REGION Network 10: DIa5
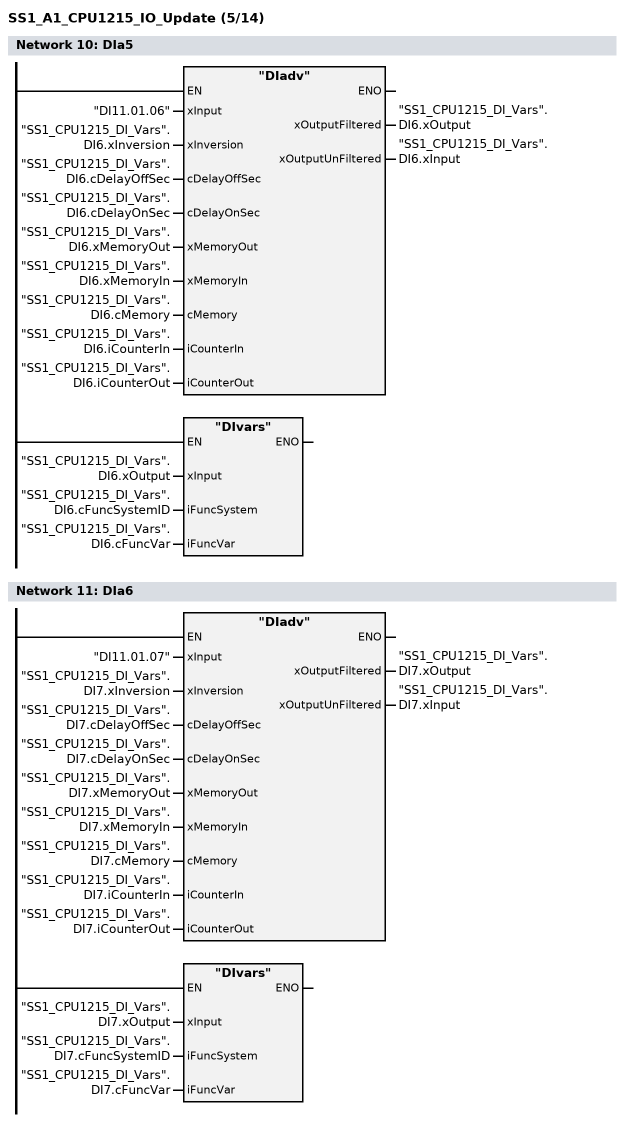
   RUNG wire#powerrail
      "DIadv"(xInput := "DI11.01.06", xInversion := "SS1_CPU1215_DI_Vars".DI6.xInversion, cDelayOffSec := "SS1_CPU1215_DI_Vars".DI6.cDelayOffSec, cDelayOnSec := "SS1_CPU1215_DI_Vars".DI6.cDelayOnSec, xMemoryOut := "SS1_CPU1215_DI_Vars".DI6.xMemoryOut, xMemoryIn := "SS1_CPU1215_DI_Vars".DI6.xMemoryIn, cMemory := "SS1_CPU1215_DI_Vars".DI6.cMemory, xOutputFiltered => "SS1_CPU1215_DI_Vars".DI6.xOutput, xOutputUnFiltered => "SS1_CPU1215_DI_Vars".DI6.xInput, iCounterIn := "SS1_CPU1215_DI_Vars".DI6.iCounterIn, iCounterOut := "SS1_CPU1215_DI_Vars".DI6.iCounterOut)
   END_RUNG
   RUNG wire#powerrail
      "DIvars"(xInput := "SS1_CPU1215_DI_Vars".DI6.xOutput, iFuncSystem := "SS1_CPU1215_DI_Vars".DI6.cFuncSystemID, iFuncVar := "SS1_CPU1215_DI_Vars".DI6.cFuncVar)
   END_RUNG
   // the same network as SCL:
   "DIadv"(xInput := "DI11.01.06",
           xInversion := "SS1_CPU1215_DI_Vars".DI6.xInversion,
           cDelayOffSec := "SS1_CPU1215_DI_Vars".DI6.cDelayOffSec,
           cDelayOnSec := "SS1_CPU1215_DI_Vars".DI6.cDelayOnSec,
           xMemoryOut := "SS1_CPU1215_DI_Vars".DI6.xMemoryOut,
           xMemoryIn := "SS1_CPU1215_DI_Vars".DI6.xMemoryIn,
           cMemory := "SS1_CPU1215_DI_Vars".DI6.cMemory,
           iCounterIn := "SS1_CPU1215_DI_Vars".DI6.iCounterIn,
           iCounterOut := "SS1_CPU1215_DI_Vars".DI6.iCounterOut,
           xOutputFiltered => "SS1_CPU1215_DI_Vars".DI6.xOutput,
           xOutputUnFiltered => "SS1_CPU1215_DI_Vars".DI6.xInput);
   "DIvars"(xInput := "SS1_CPU1215_DI_Vars".DI6.xOutput,
            iFuncSystem := "SS1_CPU1215_DI_Vars".DI6.cFuncSystemID,
            iFuncVar := "SS1_CPU1215_DI_Vars".DI6.cFuncVar);
END_REGION

REGION Network 11: DIa6
   RUNG wire#powerrail
      "DIadv"(xInput := "DI11.01.07", xInversion := "SS1_CPU1215_DI_Vars".DI7.xInversion, cDelayOffSec := "SS1_CPU1215_DI_Vars".DI7.cDelayOffSec, cDelayOnSec := "SS1_CPU1215_DI_Vars".DI7.cDelayOnSec, xMemoryOut := "SS1_CPU1215_DI_Vars".DI7.xMemoryOut, xMemoryIn := "SS1_CPU1215_DI_Vars".DI7.xMemoryIn, cMemory := "SS1_CPU1215_DI_Vars".DI7.cMemory, xOutputFiltered => "SS1_CPU1215_DI_Vars".DI7.xOutput, xOutputUnFiltered => "SS1_CPU1215_DI_Vars".DI7.xInput, iCounterIn := "SS1_CPU1215_DI_Vars".DI7.iCounterIn, iCounterOut := "SS1_CPU1215_DI_Vars".DI7.iCounterOut)
   END_RUNG
   RUNG wire#powerrail
      "DIvars"(xInput := "SS1_CPU1215_DI_Vars".DI7.xOutput, iFuncSystem := "SS1_CPU1215_DI_Vars".DI7.cFuncSystemID, iFuncVar := "SS1_CPU1215_DI_Vars".DI7.cFuncVar)
   END_RUNG
   // the same network as SCL:
   "DIadv"(xInput := "DI11.01.07",
           xInversion := "SS1_CPU1215_DI_Vars".DI7.xInversion,
           cDelayOffSec := "SS1_CPU1215_DI_Vars".DI7.cDelayOffSec,
           cDelayOnSec := "SS1_CPU1215_DI_Vars".DI7.cDelayOnSec,
           xMemoryOut := "SS1_CPU1215_DI_Vars".DI7.xMemoryOut,
           xMemoryIn := "SS1_CPU1215_DI_Vars".DI7.xMemoryIn,
           cMemory := "SS1_CPU1215_DI_Vars".DI7.cMemory,
           iCounterIn := "SS1_CPU1215_DI_Vars".DI7.iCounterIn,
           iCounterOut := "SS1_CPU1215_DI_Vars".DI7.iCounterOut,
           xOutputFiltered => "SS1_CPU1215_DI_Vars".DI7.xOutput,
           xOutputUnFiltered => "SS1_CPU1215_DI_Vars".DI7.xInput);
   "DIvars"(xInput := "SS1_CPU1215_DI_Vars".DI7.xOutput,
            iFuncSystem := "SS1_CPU1215_DI_Vars".DI7.cFuncSystemID,
            iFuncVar := "SS1_CPU1215_DI_Vars".DI7.cFuncVar);
END_REGION

REGION Network 12: DIa7 / DI01.1.08 EDP під охороною
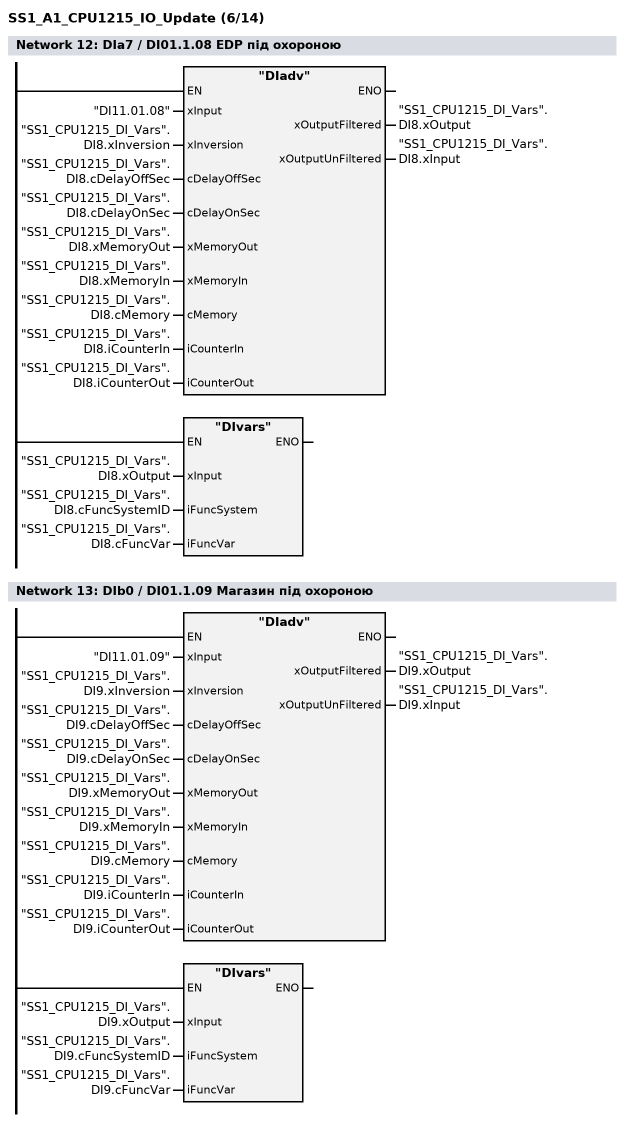
   RUNG wire#powerrail
      "DIadv"(xInput := "DI11.01.08", xInversion := "SS1_CPU1215_DI_Vars".DI8.xInversion, cDelayOffSec := "SS1_CPU1215_DI_Vars".DI8.cDelayOffSec, cDelayOnSec := "SS1_CPU1215_DI_Vars".DI8.cDelayOnSec, xMemoryOut := "SS1_CPU1215_DI_Vars".DI8.xMemoryOut, xMemoryIn := "SS1_CPU1215_DI_Vars".DI8.xMemoryIn, cMemory := "SS1_CPU1215_DI_Vars".DI8.cMemory, iCounterIn := "SS1_CPU1215_DI_Vars".DI8.iCounterIn, iCounterOut := "SS1_CPU1215_DI_Vars".DI8.iCounterOut, xOutputFiltered => "SS1_CPU1215_DI_Vars".DI8.xOutput, xOutputUnFiltered => "SS1_CPU1215_DI_Vars".DI8.xInput)
   END_RUNG
   RUNG wire#powerrail
      "DIvars"(xInput := "SS1_CPU1215_DI_Vars".DI8.xOutput, iFuncSystem := "SS1_CPU1215_DI_Vars".DI8.cFuncSystemID, iFuncVar := "SS1_CPU1215_DI_Vars".DI8.cFuncVar)
   END_RUNG
   // the same network as SCL:
   "DIadv"(xInput := "DI11.01.08",
           xInversion := "SS1_CPU1215_DI_Vars".DI8.xInversion,
           cDelayOffSec := "SS1_CPU1215_DI_Vars".DI8.cDelayOffSec,
           cDelayOnSec := "SS1_CPU1215_DI_Vars".DI8.cDelayOnSec,
           xMemoryOut := "SS1_CPU1215_DI_Vars".DI8.xMemoryOut,
           xMemoryIn := "SS1_CPU1215_DI_Vars".DI8.xMemoryIn,
           cMemory := "SS1_CPU1215_DI_Vars".DI8.cMemory,
           iCounterIn := "SS1_CPU1215_DI_Vars".DI8.iCounterIn,
           iCounterOut := "SS1_CPU1215_DI_Vars".DI8.iCounterOut,
           xOutputFiltered => "SS1_CPU1215_DI_Vars".DI8.xOutput,
           xOutputUnFiltered => "SS1_CPU1215_DI_Vars".DI8.xInput);
   "DIvars"(xInput := "SS1_CPU1215_DI_Vars".DI8.xOutput,
            iFuncSystem := "SS1_CPU1215_DI_Vars".DI8.cFuncSystemID,
            iFuncVar := "SS1_CPU1215_DI_Vars".DI8.cFuncVar);
END_REGION

REGION Network 13: DIb0 / DI01.1.09 Магазин під охороною
   RUNG wire#powerrail
      "DIadv"(xInput := "DI11.01.09", xInversion := "SS1_CPU1215_DI_Vars".DI9.xInversion, cDelayOffSec := "SS1_CPU1215_DI_Vars".DI9.cDelayOffSec, cDelayOnSec := "SS1_CPU1215_DI_Vars".DI9.cDelayOnSec, xMemoryOut := "SS1_CPU1215_DI_Vars".DI9.xMemoryOut, xMemoryIn := "SS1_CPU1215_DI_Vars".DI9.xMemoryIn, cMemory := "SS1_CPU1215_DI_Vars".DI9.cMemory, xOutputFiltered => "SS1_CPU1215_DI_Vars".DI9.xOutput, xOutputUnFiltered => "SS1_CPU1215_DI_Vars".DI9.xInput, iCounterIn := "SS1_CPU1215_DI_Vars".DI9.iCounterIn, iCounterOut := "SS1_CPU1215_DI_Vars".DI9.iCounterOut)
   END_RUNG
   RUNG wire#powerrail
      "DIvars"(xInput := "SS1_CPU1215_DI_Vars".DI9.xOutput, iFuncSystem := "SS1_CPU1215_DI_Vars".DI9.cFuncSystemID, iFuncVar := "SS1_CPU1215_DI_Vars".DI9.cFuncVar)
   END_RUNG
   // the same network as SCL:
   "DIadv"(xInput := "DI11.01.09",
           xInversion := "SS1_CPU1215_DI_Vars".DI9.xInversion,
           cDelayOffSec := "SS1_CPU1215_DI_Vars".DI9.cDelayOffSec,
           cDelayOnSec := "SS1_CPU1215_DI_Vars".DI9.cDelayOnSec,
           xMemoryOut := "SS1_CPU1215_DI_Vars".DI9.xMemoryOut,
           xMemoryIn := "SS1_CPU1215_DI_Vars".DI9.xMemoryIn,
           cMemory := "SS1_CPU1215_DI_Vars".DI9.cMemory,
           iCounterIn := "SS1_CPU1215_DI_Vars".DI9.iCounterIn,
           iCounterOut := "SS1_CPU1215_DI_Vars".DI9.iCounterOut,
           xOutputFiltered => "SS1_CPU1215_DI_Vars".DI9.xOutput,
           xOutputUnFiltered => "SS1_CPU1215_DI_Vars".DI9.xInput);
   "DIvars"(xInput := "SS1_CPU1215_DI_Vars".DI9.xOutput,
            iFuncSystem := "SS1_CPU1215_DI_Vars".DI9.cFuncSystemID,
            iFuncVar := "SS1_CPU1215_DI_Vars".DI9.cFuncVar);
END_REGION

REGION Network 14: DIb1 / DI01.1.10 Аварійний рівень загазованості
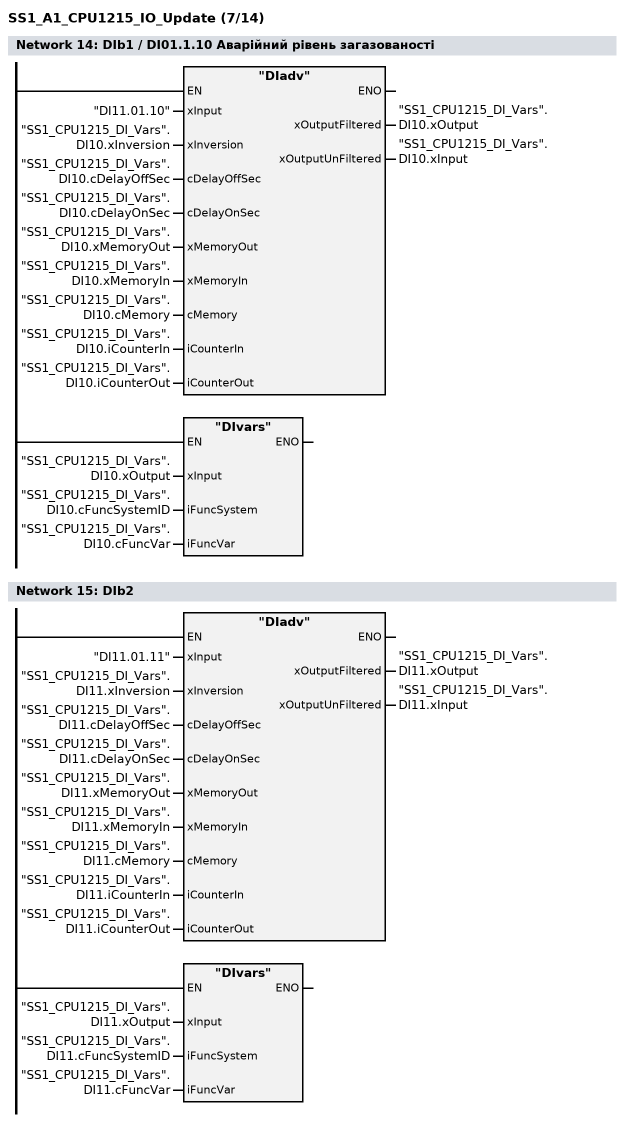
   RUNG wire#powerrail
      "DIadv"(xInput := "DI11.01.10", xInversion := "SS1_CPU1215_DI_Vars".DI10.xInversion, cDelayOffSec := "SS1_CPU1215_DI_Vars".DI10.cDelayOffSec, cDelayOnSec := "SS1_CPU1215_DI_Vars".DI10.cDelayOnSec, xMemoryOut := "SS1_CPU1215_DI_Vars".DI10.xMemoryOut, xMemoryIn := "SS1_CPU1215_DI_Vars".DI10.xMemoryIn, cMemory := "SS1_CPU1215_DI_Vars".DI10.cMemory, xOutputFiltered => "SS1_CPU1215_DI_Vars".DI10.xOutput, xOutputUnFiltered => "SS1_CPU1215_DI_Vars".DI10.xInput, iCounterIn := "SS1_CPU1215_DI_Vars".DI10.iCounterIn, iCounterOut := "SS1_CPU1215_DI_Vars".DI10.iCounterOut)
   END_RUNG
   RUNG wire#powerrail
      "DIvars"(xInput := "SS1_CPU1215_DI_Vars".DI10.xOutput, iFuncSystem := "SS1_CPU1215_DI_Vars".DI10.cFuncSystemID, iFuncVar := "SS1_CPU1215_DI_Vars".DI10.cFuncVar)
   END_RUNG
   // the same network as SCL:
   "DIadv"(xInput := "DI11.01.10",
           xInversion := "SS1_CPU1215_DI_Vars".DI10.xInversion,
           cDelayOffSec := "SS1_CPU1215_DI_Vars".DI10.cDelayOffSec,
           cDelayOnSec := "SS1_CPU1215_DI_Vars".DI10.cDelayOnSec,
           xMemoryOut := "SS1_CPU1215_DI_Vars".DI10.xMemoryOut,
           xMemoryIn := "SS1_CPU1215_DI_Vars".DI10.xMemoryIn,
           cMemory := "SS1_CPU1215_DI_Vars".DI10.cMemory,
           iCounterIn := "SS1_CPU1215_DI_Vars".DI10.iCounterIn,
           iCounterOut := "SS1_CPU1215_DI_Vars".DI10.iCounterOut,
           xOutputFiltered => "SS1_CPU1215_DI_Vars".DI10.xOutput,
           xOutputUnFiltered => "SS1_CPU1215_DI_Vars".DI10.xInput);
   "DIvars"(xInput := "SS1_CPU1215_DI_Vars".DI10.xOutput,
            iFuncSystem := "SS1_CPU1215_DI_Vars".DI10.cFuncSystemID,
            iFuncVar := "SS1_CPU1215_DI_Vars".DI10.cFuncVar);
END_REGION

REGION Network 15: DIb2
   RUNG wire#powerrail
      "DIadv"(xInput := "DI11.01.11", xInversion := "SS1_CPU1215_DI_Vars".DI11.xInversion, cDelayOffSec := "SS1_CPU1215_DI_Vars".DI11.cDelayOffSec, cDelayOnSec := "SS1_CPU1215_DI_Vars".DI11.cDelayOnSec, xMemoryOut := "SS1_CPU1215_DI_Vars".DI11.xMemoryOut, xMemoryIn := "SS1_CPU1215_DI_Vars".DI11.xMemoryIn, cMemory := "SS1_CPU1215_DI_Vars".DI11.cMemory, iCounterIn := "SS1_CPU1215_DI_Vars".DI11.iCounterIn, iCounterOut := "SS1_CPU1215_DI_Vars".DI11.iCounterOut, xOutputFiltered => "SS1_CPU1215_DI_Vars".DI11.xOutput, xOutputUnFiltered => "SS1_CPU1215_DI_Vars".DI11.xInput)
   END_RUNG
   RUNG wire#powerrail
      "DIvars"(xInput := "SS1_CPU1215_DI_Vars".DI11.xOutput, iFuncSystem := "SS1_CPU1215_DI_Vars".DI11.cFuncSystemID, iFuncVar := "SS1_CPU1215_DI_Vars".DI11.cFuncVar)
   END_RUNG
   // the same network as SCL:
   "DIadv"(xInput := "DI11.01.11",
           xInversion := "SS1_CPU1215_DI_Vars".DI11.xInversion,
           cDelayOffSec := "SS1_CPU1215_DI_Vars".DI11.cDelayOffSec,
           cDelayOnSec := "SS1_CPU1215_DI_Vars".DI11.cDelayOnSec,
           xMemoryOut := "SS1_CPU1215_DI_Vars".DI11.xMemoryOut,
           xMemoryIn := "SS1_CPU1215_DI_Vars".DI11.xMemoryIn,
           cMemory := "SS1_CPU1215_DI_Vars".DI11.cMemory,
           iCounterIn := "SS1_CPU1215_DI_Vars".DI11.iCounterIn,
           iCounterOut := "SS1_CPU1215_DI_Vars".DI11.iCounterOut,
           xOutputFiltered => "SS1_CPU1215_DI_Vars".DI11.xOutput,
           xOutputUnFiltered => "SS1_CPU1215_DI_Vars".DI11.xInput);
   "DIvars"(xInput := "SS1_CPU1215_DI_Vars".DI11.xOutput,
            iFuncSystem := "SS1_CPU1215_DI_Vars".DI11.cFuncSystemID,
            iFuncVar := "SS1_CPU1215_DI_Vars".DI11.cFuncVar);
END_REGION

REGION Network 16: DIb3
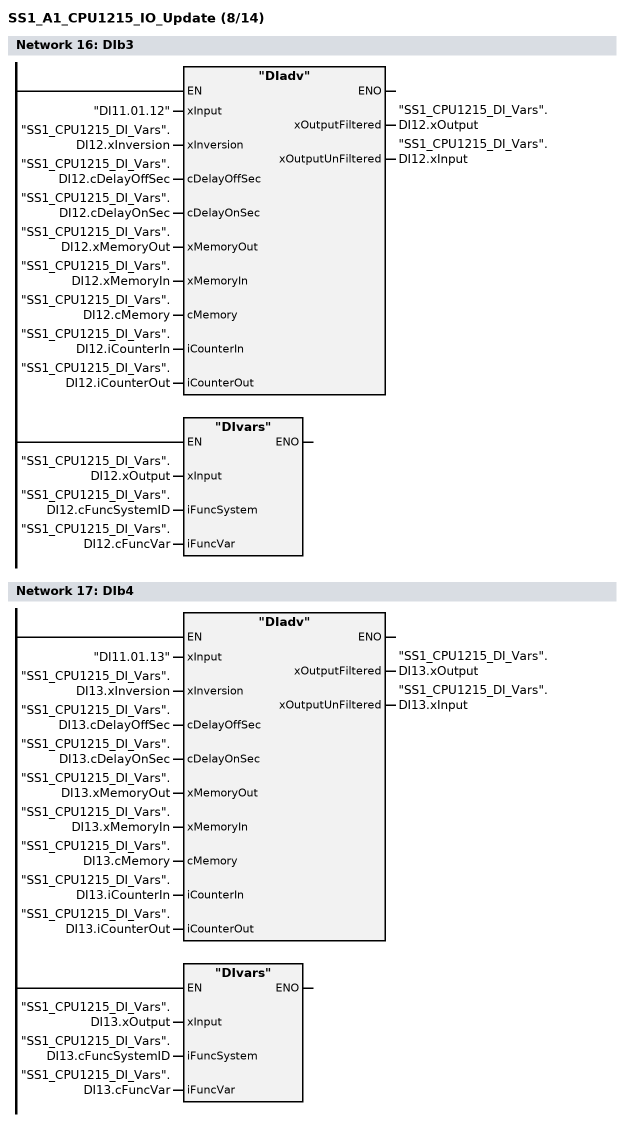
   RUNG wire#powerrail
      "DIadv"(xInput := "DI11.01.12", xInversion := "SS1_CPU1215_DI_Vars".DI12.xInversion, cDelayOffSec := "SS1_CPU1215_DI_Vars".DI12.cDelayOffSec, cDelayOnSec := "SS1_CPU1215_DI_Vars".DI12.cDelayOnSec, xMemoryOut := "SS1_CPU1215_DI_Vars".DI12.xMemoryOut, xMemoryIn := "SS1_CPU1215_DI_Vars".DI12.xMemoryIn, cMemory := "SS1_CPU1215_DI_Vars".DI12.cMemory, xOutputFiltered => "SS1_CPU1215_DI_Vars".DI12.xOutput, xOutputUnFiltered => "SS1_CPU1215_DI_Vars".DI12.xInput, iCounterIn := "SS1_CPU1215_DI_Vars".DI12.iCounterIn, iCounterOut := "SS1_CPU1215_DI_Vars".DI12.iCounterOut)
   END_RUNG
   RUNG wire#powerrail
      "DIvars"(xInput := "SS1_CPU1215_DI_Vars".DI12.xOutput, iFuncSystem := "SS1_CPU1215_DI_Vars".DI12.cFuncSystemID, iFuncVar := "SS1_CPU1215_DI_Vars".DI12.cFuncVar)
   END_RUNG
   // the same network as SCL:
   "DIadv"(xInput := "DI11.01.12",
           xInversion := "SS1_CPU1215_DI_Vars".DI12.xInversion,
           cDelayOffSec := "SS1_CPU1215_DI_Vars".DI12.cDelayOffSec,
           cDelayOnSec := "SS1_CPU1215_DI_Vars".DI12.cDelayOnSec,
           xMemoryOut := "SS1_CPU1215_DI_Vars".DI12.xMemoryOut,
           xMemoryIn := "SS1_CPU1215_DI_Vars".DI12.xMemoryIn,
           cMemory := "SS1_CPU1215_DI_Vars".DI12.cMemory,
           iCounterIn := "SS1_CPU1215_DI_Vars".DI12.iCounterIn,
           iCounterOut := "SS1_CPU1215_DI_Vars".DI12.iCounterOut,
           xOutputFiltered => "SS1_CPU1215_DI_Vars".DI12.xOutput,
           xOutputUnFiltered => "SS1_CPU1215_DI_Vars".DI12.xInput);
   "DIvars"(xInput := "SS1_CPU1215_DI_Vars".DI12.xOutput,
            iFuncSystem := "SS1_CPU1215_DI_Vars".DI12.cFuncSystemID,
            iFuncVar := "SS1_CPU1215_DI_Vars".DI12.cFuncVar);
END_REGION

REGION Network 17: DIb4
   RUNG wire#powerrail
      "DIadv"(xInput := "DI11.01.13", xInversion := "SS1_CPU1215_DI_Vars".DI13.xInversion, cDelayOffSec := "SS1_CPU1215_DI_Vars".DI13.cDelayOffSec, cDelayOnSec := "SS1_CPU1215_DI_Vars".DI13.cDelayOnSec, xMemoryOut := "SS1_CPU1215_DI_Vars".DI13.xMemoryOut, xMemoryIn := "SS1_CPU1215_DI_Vars".DI13.xMemoryIn, cMemory := "SS1_CPU1215_DI_Vars".DI13.cMemory, xOutputFiltered => "SS1_CPU1215_DI_Vars".DI13.xOutput, xOutputUnFiltered => "SS1_CPU1215_DI_Vars".DI13.xInput, iCounterIn := "SS1_CPU1215_DI_Vars".DI13.iCounterIn, iCounterOut := "SS1_CPU1215_DI_Vars".DI13.iCounterOut)
   END_RUNG
   RUNG wire#powerrail
      "DIvars"(xInput := "SS1_CPU1215_DI_Vars".DI13.xOutput, iFuncSystem := "SS1_CPU1215_DI_Vars".DI13.cFuncSystemID, iFuncVar := "SS1_CPU1215_DI_Vars".DI13.cFuncVar)
   END_RUNG
   // the same network as SCL:
   "DIadv"(xInput := "DI11.01.13",
           xInversion := "SS1_CPU1215_DI_Vars".DI13.xInversion,
           cDelayOffSec := "SS1_CPU1215_DI_Vars".DI13.cDelayOffSec,
           cDelayOnSec := "SS1_CPU1215_DI_Vars".DI13.cDelayOnSec,
           xMemoryOut := "SS1_CPU1215_DI_Vars".DI13.xMemoryOut,
           xMemoryIn := "SS1_CPU1215_DI_Vars".DI13.xMemoryIn,
           cMemory := "SS1_CPU1215_DI_Vars".DI13.cMemory,
           iCounterIn := "SS1_CPU1215_DI_Vars".DI13.iCounterIn,
           iCounterOut := "SS1_CPU1215_DI_Vars".DI13.iCounterOut,
           xOutputFiltered => "SS1_CPU1215_DI_Vars".DI13.xOutput,
           xOutputUnFiltered => "SS1_CPU1215_DI_Vars".DI13.xInput);
   "DIvars"(xInput := "SS1_CPU1215_DI_Vars".DI13.xOutput,
            iFuncSystem := "SS1_CPU1215_DI_Vars".DI13.cFuncSystemID,
            iFuncVar := "SS1_CPU1215_DI_Vars".DI13.cFuncVar);
END_REGION

REGION Network 18: DIb5 / DI01.1.14 Спрацювання охоронної сигналізації
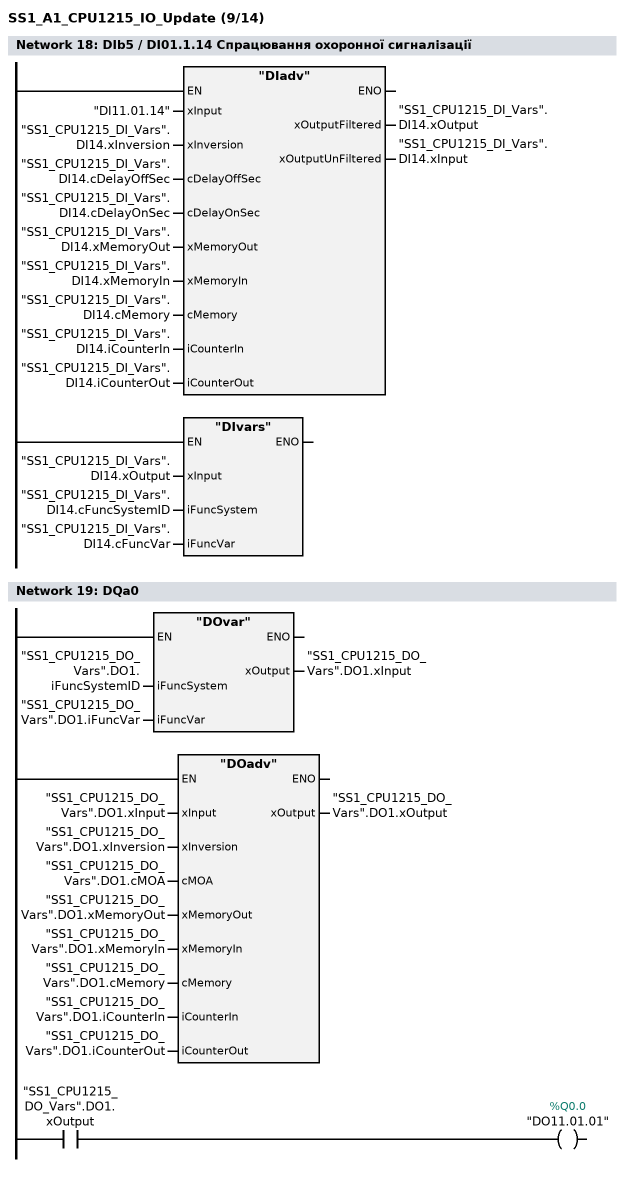
   RUNG wire#powerrail
      "DIadv"(xInput := "DI11.01.14", xInversion := "SS1_CPU1215_DI_Vars".DI14.xInversion, cDelayOffSec := "SS1_CPU1215_DI_Vars".DI14.cDelayOffSec, cDelayOnSec := "SS1_CPU1215_DI_Vars".DI14.cDelayOnSec, xMemoryOut := "SS1_CPU1215_DI_Vars".DI14.xMemoryOut, xMemoryIn := "SS1_CPU1215_DI_Vars".DI14.xMemoryIn, cMemory := "SS1_CPU1215_DI_Vars".DI14.cMemory, xOutputFiltered => "SS1_CPU1215_DI_Vars".DI14.xOutput, xOutputUnFiltered => "SS1_CPU1215_DI_Vars".DI14.xInput, iCounterIn := "SS1_CPU1215_DI_Vars".DI14.iCounterIn, iCounterOut := "SS1_CPU1215_DI_Vars".DI14.iCounterOut)
   END_RUNG
   RUNG wire#powerrail
      "DIvars"(xInput := "SS1_CPU1215_DI_Vars".DI14.xOutput, iFuncSystem := "SS1_CPU1215_DI_Vars".DI14.cFuncSystemID, iFuncVar := "SS1_CPU1215_DI_Vars".DI14.cFuncVar)
   END_RUNG
   // the same network as SCL:
   "DIadv"(xInput := "DI11.01.14",
           xInversion := "SS1_CPU1215_DI_Vars".DI14.xInversion,
           cDelayOffSec := "SS1_CPU1215_DI_Vars".DI14.cDelayOffSec,
           cDelayOnSec := "SS1_CPU1215_DI_Vars".DI14.cDelayOnSec,
           xMemoryOut := "SS1_CPU1215_DI_Vars".DI14.xMemoryOut,
           xMemoryIn := "SS1_CPU1215_DI_Vars".DI14.xMemoryIn,
           cMemory := "SS1_CPU1215_DI_Vars".DI14.cMemory,
           iCounterIn := "SS1_CPU1215_DI_Vars".DI14.iCounterIn,
           iCounterOut := "SS1_CPU1215_DI_Vars".DI14.iCounterOut,
           xOutputFiltered => "SS1_CPU1215_DI_Vars".DI14.xOutput,
           xOutputUnFiltered => "SS1_CPU1215_DI_Vars".DI14.xInput);
   "DIvars"(xInput := "SS1_CPU1215_DI_Vars".DI14.xOutput,
            iFuncSystem := "SS1_CPU1215_DI_Vars".DI14.cFuncSystemID,
            iFuncVar := "SS1_CPU1215_DI_Vars".DI14.cFuncVar);
END_REGION

REGION Network 19: DQa0
   RUNG wire#powerrail
      "DOvar"(iFuncSystem := "SS1_CPU1215_DO_Vars".DO1.iFuncSystemID, iFuncVar := "SS1_CPU1215_DO_Vars".DO1.iFuncVar, xOutput => "SS1_CPU1215_DO_Vars".DO1.xInput)
   END_RUNG
   RUNG wire#powerrail
      "DOadv"(xInput := "SS1_CPU1215_DO_Vars".DO1.xInput, xInversion := "SS1_CPU1215_DO_Vars".DO1.xInversion, cMOA := "SS1_CPU1215_DO_Vars".DO1.cMOA, xMemoryOut := "SS1_CPU1215_DO_Vars".DO1.xMemoryOut, xMemoryIn := "SS1_CPU1215_DO_Vars".DO1.xMemoryIn, cMemory := "SS1_CPU1215_DO_Vars".DO1.cMemory, xOutput => "SS1_CPU1215_DO_Vars".DO1.xOutput, iCounterIn := "SS1_CPU1215_DO_Vars".DO1.iCounterIn, iCounterOut := "SS1_CPU1215_DO_Vars".DO1.iCounterOut)
   END_RUNG
   RUNG wire#powerrail
      Contact( "SS1_CPU1215_DO_Vars".DO1.xOutput )
      Coil( "DO11.01.01" )
   END_RUNG
   // the same network as SCL:
   "DOvar"(iFuncSystem := "SS1_CPU1215_DO_Vars".DO1.iFuncSystemID,
           iFuncVar := "SS1_CPU1215_DO_Vars".DO1.iFuncVar,
           xOutput => "SS1_CPU1215_DO_Vars".DO1.xInput);
   "DOadv"(xInput := "SS1_CPU1215_DO_Vars".DO1.xInput,
           xInversion := "SS1_CPU1215_DO_Vars".DO1.xInversion,
           cMOA := "SS1_CPU1215_DO_Vars".DO1.cMOA,
           xMemoryOut := "SS1_CPU1215_DO_Vars".DO1.xMemoryOut,
           xMemoryIn := "SS1_CPU1215_DO_Vars".DO1.xMemoryIn,
           cMemory := "SS1_CPU1215_DO_Vars".DO1.cMemory,
           iCounterIn := "SS1_CPU1215_DO_Vars".DO1.iCounterIn,
           iCounterOut := "SS1_CPU1215_DO_Vars".DO1.iCounterOut,
           xOutput => "SS1_CPU1215_DO_Vars".DO1.xOutput);
   "DO11.01.01" := "SS1_CPU1215_DO_Vars".DO1.xOutput;
END_REGION

REGION Network 20: DQa1
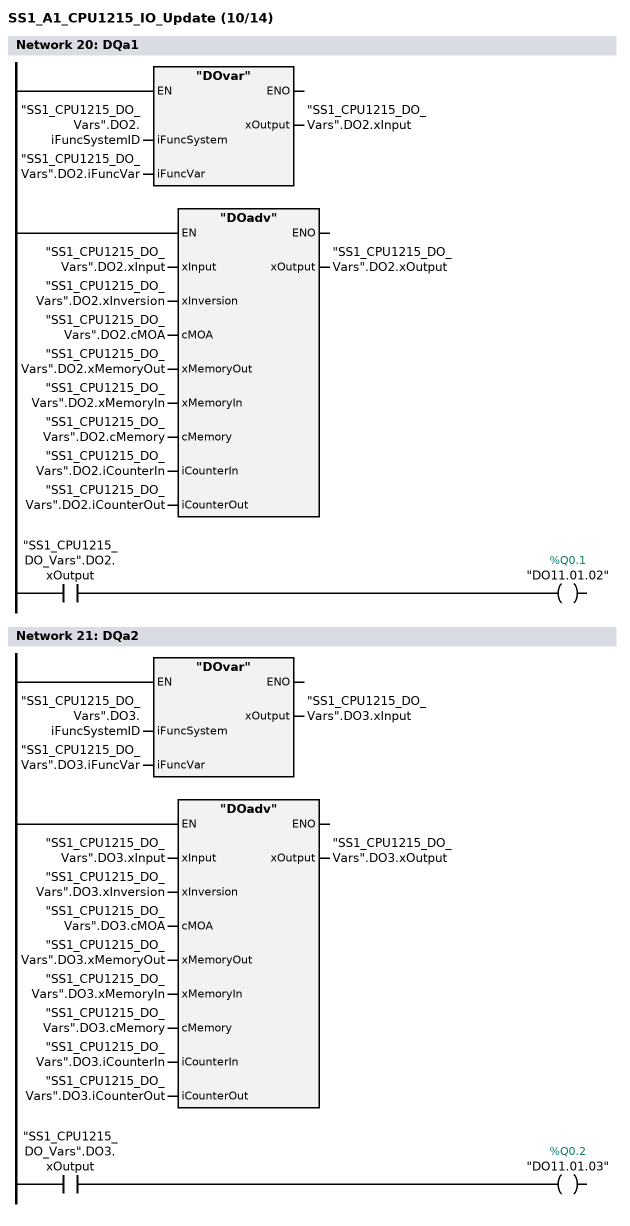
   RUNG wire#powerrail
      "DOvar"(iFuncSystem := "SS1_CPU1215_DO_Vars".DO2.iFuncSystemID, iFuncVar := "SS1_CPU1215_DO_Vars".DO2.iFuncVar, xOutput => "SS1_CPU1215_DO_Vars".DO2.xInput)
   END_RUNG
   RUNG wire#powerrail
      "DOadv"(xInput := "SS1_CPU1215_DO_Vars".DO2.xInput, xInversion := "SS1_CPU1215_DO_Vars".DO2.xInversion, cMOA := "SS1_CPU1215_DO_Vars".DO2.cMOA, xMemoryOut := "SS1_CPU1215_DO_Vars".DO2.xMemoryOut, xMemoryIn := "SS1_CPU1215_DO_Vars".DO2.xMemoryIn, cMemory := "SS1_CPU1215_DO_Vars".DO2.cMemory, xOutput => "SS1_CPU1215_DO_Vars".DO2.xOutput, iCounterIn := "SS1_CPU1215_DO_Vars".DO2.iCounterIn, iCounterOut := "SS1_CPU1215_DO_Vars".DO2.iCounterOut)
   END_RUNG
   RUNG wire#powerrail
      Contact( "SS1_CPU1215_DO_Vars".DO2.xOutput )
      Coil( "DO11.01.02" )
   END_RUNG
   // the same network as SCL:
   "DOvar"(iFuncSystem := "SS1_CPU1215_DO_Vars".DO2.iFuncSystemID,
           iFuncVar := "SS1_CPU1215_DO_Vars".DO2.iFuncVar,
           xOutput => "SS1_CPU1215_DO_Vars".DO2.xInput);
   "DOadv"(xInput := "SS1_CPU1215_DO_Vars".DO2.xInput,
           xInversion := "SS1_CPU1215_DO_Vars".DO2.xInversion,
           cMOA := "SS1_CPU1215_DO_Vars".DO2.cMOA,
           xMemoryOut := "SS1_CPU1215_DO_Vars".DO2.xMemoryOut,
           xMemoryIn := "SS1_CPU1215_DO_Vars".DO2.xMemoryIn,
           cMemory := "SS1_CPU1215_DO_Vars".DO2.cMemory,
           iCounterIn := "SS1_CPU1215_DO_Vars".DO2.iCounterIn,
           iCounterOut := "SS1_CPU1215_DO_Vars".DO2.iCounterOut,
           xOutput => "SS1_CPU1215_DO_Vars".DO2.xOutput);
   "DO11.01.02" := "SS1_CPU1215_DO_Vars".DO2.xOutput;
END_REGION

REGION Network 21: DQa2
   RUNG wire#powerrail
      "DOvar"(iFuncSystem := "SS1_CPU1215_DO_Vars".DO3.iFuncSystemID, iFuncVar := "SS1_CPU1215_DO_Vars".DO3.iFuncVar, xOutput => "SS1_CPU1215_DO_Vars".DO3.xInput)
   END_RUNG
   RUNG wire#powerrail
      "DOadv"(xInput := "SS1_CPU1215_DO_Vars".DO3.xInput, xInversion := "SS1_CPU1215_DO_Vars".DO3.xInversion, cMOA := "SS1_CPU1215_DO_Vars".DO3.cMOA, xMemoryOut := "SS1_CPU1215_DO_Vars".DO3.xMemoryOut, xMemoryIn := "SS1_CPU1215_DO_Vars".DO3.xMemoryIn, cMemory := "SS1_CPU1215_DO_Vars".DO3.cMemory, xOutput => "SS1_CPU1215_DO_Vars".DO3.xOutput, iCounterIn := "SS1_CPU1215_DO_Vars".DO3.iCounterIn, iCounterOut := "SS1_CPU1215_DO_Vars".DO3.iCounterOut)
   END_RUNG
   RUNG wire#powerrail
      Contact( "SS1_CPU1215_DO_Vars".DO3.xOutput )
      Coil( "DO11.01.03" )
   END_RUNG
   // the same network as SCL:
   "DOvar"(iFuncSystem := "SS1_CPU1215_DO_Vars".DO3.iFuncSystemID,
           iFuncVar := "SS1_CPU1215_DO_Vars".DO3.iFuncVar,
           xOutput => "SS1_CPU1215_DO_Vars".DO3.xInput);
   "DOadv"(xInput := "SS1_CPU1215_DO_Vars".DO3.xInput,
           xInversion := "SS1_CPU1215_DO_Vars".DO3.xInversion,
           cMOA := "SS1_CPU1215_DO_Vars".DO3.cMOA,
           xMemoryOut := "SS1_CPU1215_DO_Vars".DO3.xMemoryOut,
           xMemoryIn := "SS1_CPU1215_DO_Vars".DO3.xMemoryIn,
           cMemory := "SS1_CPU1215_DO_Vars".DO3.cMemory,
           iCounterIn := "SS1_CPU1215_DO_Vars".DO3.iCounterIn,
           iCounterOut := "SS1_CPU1215_DO_Vars".DO3.iCounterOut,
           xOutput => "SS1_CPU1215_DO_Vars".DO3.xOutput);
   "DO11.01.03" := "SS1_CPU1215_DO_Vars".DO3.xOutput;
END_REGION

REGION Network 22: DQa3
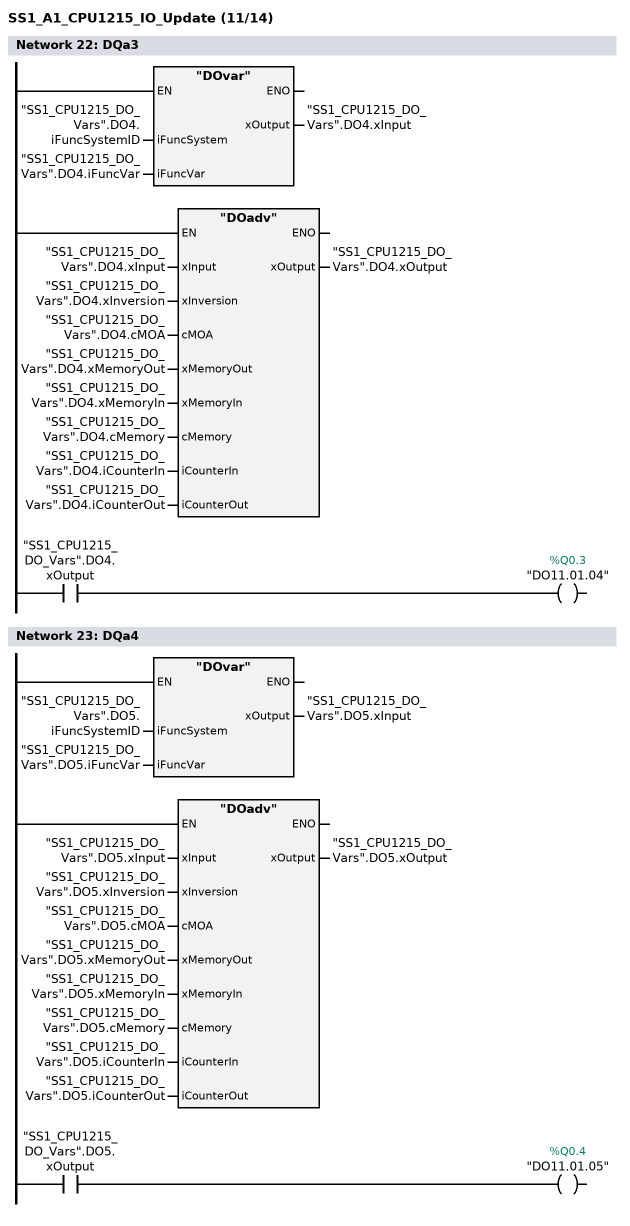
   RUNG wire#powerrail
      "DOvar"(iFuncSystem := "SS1_CPU1215_DO_Vars".DO4.iFuncSystemID, iFuncVar := "SS1_CPU1215_DO_Vars".DO4.iFuncVar, xOutput => "SS1_CPU1215_DO_Vars".DO4.xInput)
   END_RUNG
   RUNG wire#powerrail
      "DOadv"(xInput := "SS1_CPU1215_DO_Vars".DO4.xInput, xInversion := "SS1_CPU1215_DO_Vars".DO4.xInversion, cMOA := "SS1_CPU1215_DO_Vars".DO4.cMOA, xMemoryOut := "SS1_CPU1215_DO_Vars".DO4.xMemoryOut, xMemoryIn := "SS1_CPU1215_DO_Vars".DO4.xMemoryIn, cMemory := "SS1_CPU1215_DO_Vars".DO4.cMemory, xOutput => "SS1_CPU1215_DO_Vars".DO4.xOutput, iCounterIn := "SS1_CPU1215_DO_Vars".DO4.iCounterIn, iCounterOut := "SS1_CPU1215_DO_Vars".DO4.iCounterOut)
   END_RUNG
   RUNG wire#powerrail
      Contact( "SS1_CPU1215_DO_Vars".DO4.xOutput )
      Coil( "DO11.01.04" )
   END_RUNG
   // the same network as SCL:
   "DOvar"(iFuncSystem := "SS1_CPU1215_DO_Vars".DO4.iFuncSystemID,
           iFuncVar := "SS1_CPU1215_DO_Vars".DO4.iFuncVar,
           xOutput => "SS1_CPU1215_DO_Vars".DO4.xInput);
   "DOadv"(xInput := "SS1_CPU1215_DO_Vars".DO4.xInput,
           xInversion := "SS1_CPU1215_DO_Vars".DO4.xInversion,
           cMOA := "SS1_CPU1215_DO_Vars".DO4.cMOA,
           xMemoryOut := "SS1_CPU1215_DO_Vars".DO4.xMemoryOut,
           xMemoryIn := "SS1_CPU1215_DO_Vars".DO4.xMemoryIn,
           cMemory := "SS1_CPU1215_DO_Vars".DO4.cMemory,
           iCounterIn := "SS1_CPU1215_DO_Vars".DO4.iCounterIn,
           iCounterOut := "SS1_CPU1215_DO_Vars".DO4.iCounterOut,
           xOutput => "SS1_CPU1215_DO_Vars".DO4.xOutput);
   "DO11.01.04" := "SS1_CPU1215_DO_Vars".DO4.xOutput;
END_REGION

REGION Network 23: DQa4
   RUNG wire#powerrail
      "DOvar"(iFuncSystem := "SS1_CPU1215_DO_Vars".DO5.iFuncSystemID, iFuncVar := "SS1_CPU1215_DO_Vars".DO5.iFuncVar, xOutput => "SS1_CPU1215_DO_Vars".DO5.xInput)
   END_RUNG
   RUNG wire#powerrail
      "DOadv"(xInput := "SS1_CPU1215_DO_Vars".DO5.xInput, xInversion := "SS1_CPU1215_DO_Vars".DO5.xInversion, cMOA := "SS1_CPU1215_DO_Vars".DO5.cMOA, xMemoryOut := "SS1_CPU1215_DO_Vars".DO5.xMemoryOut, xMemoryIn := "SS1_CPU1215_DO_Vars".DO5.xMemoryIn, cMemory := "SS1_CPU1215_DO_Vars".DO5.cMemory, xOutput => "SS1_CPU1215_DO_Vars".DO5.xOutput, iCounterIn := "SS1_CPU1215_DO_Vars".DO5.iCounterIn, iCounterOut := "SS1_CPU1215_DO_Vars".DO5.iCounterOut)
   END_RUNG
   RUNG wire#powerrail
      Contact( "SS1_CPU1215_DO_Vars".DO5.xOutput )
      Coil( "DO11.01.05" )
   END_RUNG
   // the same network as SCL:
   "DOvar"(iFuncSystem := "SS1_CPU1215_DO_Vars".DO5.iFuncSystemID,
           iFuncVar := "SS1_CPU1215_DO_Vars".DO5.iFuncVar,
           xOutput => "SS1_CPU1215_DO_Vars".DO5.xInput);
   "DOadv"(xInput := "SS1_CPU1215_DO_Vars".DO5.xInput,
           xInversion := "SS1_CPU1215_DO_Vars".DO5.xInversion,
           cMOA := "SS1_CPU1215_DO_Vars".DO5.cMOA,
           xMemoryOut := "SS1_CPU1215_DO_Vars".DO5.xMemoryOut,
           xMemoryIn := "SS1_CPU1215_DO_Vars".DO5.xMemoryIn,
           cMemory := "SS1_CPU1215_DO_Vars".DO5.cMemory,
           iCounterIn := "SS1_CPU1215_DO_Vars".DO5.iCounterIn,
           iCounterOut := "SS1_CPU1215_DO_Vars".DO5.iCounterOut,
           xOutput => "SS1_CPU1215_DO_Vars".DO5.xOutput);
   "DO11.01.05" := "SS1_CPU1215_DO_Vars".DO5.xOutput;
END_REGION

REGION Network 24: DQa5
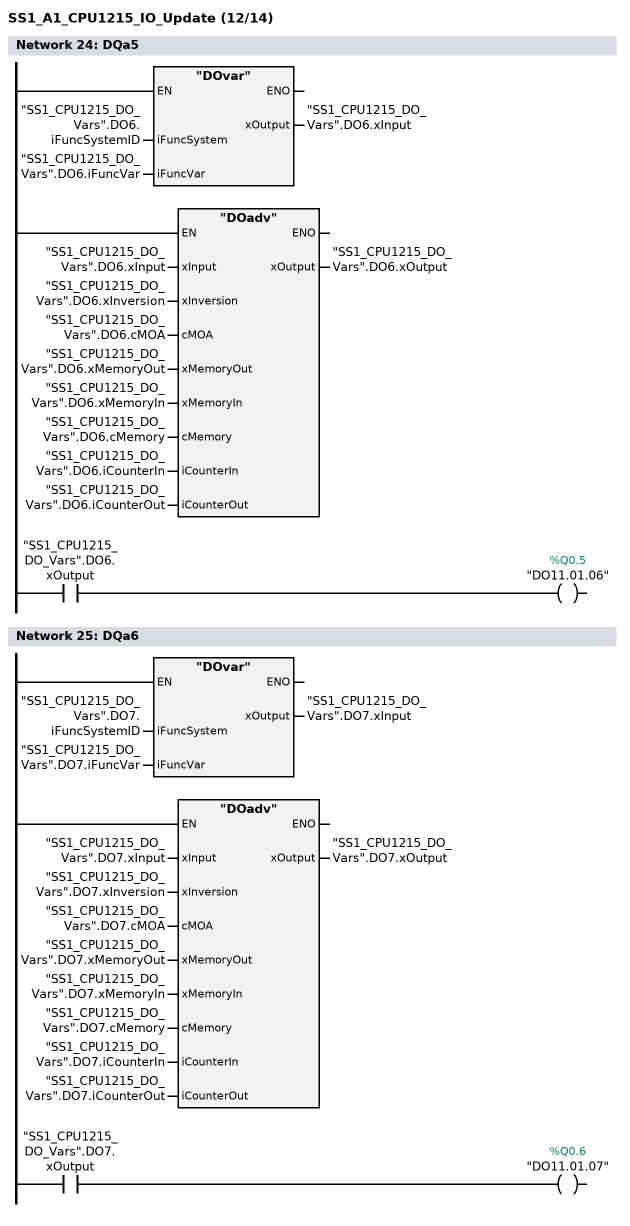
   RUNG wire#powerrail
      "DOvar"(iFuncSystem := "SS1_CPU1215_DO_Vars".DO6.iFuncSystemID, iFuncVar := "SS1_CPU1215_DO_Vars".DO6.iFuncVar, xOutput => "SS1_CPU1215_DO_Vars".DO6.xInput)
   END_RUNG
   RUNG wire#powerrail
      "DOadv"(xInput := "SS1_CPU1215_DO_Vars".DO6.xInput, xInversion := "SS1_CPU1215_DO_Vars".DO6.xInversion, cMOA := "SS1_CPU1215_DO_Vars".DO6.cMOA, xMemoryOut := "SS1_CPU1215_DO_Vars".DO6.xMemoryOut, xMemoryIn := "SS1_CPU1215_DO_Vars".DO6.xMemoryIn, cMemory := "SS1_CPU1215_DO_Vars".DO6.cMemory, xOutput => "SS1_CPU1215_DO_Vars".DO6.xOutput, iCounterIn := "SS1_CPU1215_DO_Vars".DO6.iCounterIn, iCounterOut := "SS1_CPU1215_DO_Vars".DO6.iCounterOut)
   END_RUNG
   RUNG wire#powerrail
      Contact( "SS1_CPU1215_DO_Vars".DO6.xOutput )
      Coil( "DO11.01.06" )
   END_RUNG
   // the same network as SCL:
   "DOvar"(iFuncSystem := "SS1_CPU1215_DO_Vars".DO6.iFuncSystemID,
           iFuncVar := "SS1_CPU1215_DO_Vars".DO6.iFuncVar,
           xOutput => "SS1_CPU1215_DO_Vars".DO6.xInput);
   "DOadv"(xInput := "SS1_CPU1215_DO_Vars".DO6.xInput,
           xInversion := "SS1_CPU1215_DO_Vars".DO6.xInversion,
           cMOA := "SS1_CPU1215_DO_Vars".DO6.cMOA,
           xMemoryOut := "SS1_CPU1215_DO_Vars".DO6.xMemoryOut,
           xMemoryIn := "SS1_CPU1215_DO_Vars".DO6.xMemoryIn,
           cMemory := "SS1_CPU1215_DO_Vars".DO6.cMemory,
           iCounterIn := "SS1_CPU1215_DO_Vars".DO6.iCounterIn,
           iCounterOut := "SS1_CPU1215_DO_Vars".DO6.iCounterOut,
           xOutput => "SS1_CPU1215_DO_Vars".DO6.xOutput);
   "DO11.01.06" := "SS1_CPU1215_DO_Vars".DO6.xOutput;
END_REGION

REGION Network 25: DQa6
   RUNG wire#powerrail
      "DOvar"(iFuncSystem := "SS1_CPU1215_DO_Vars".DO7.iFuncSystemID, iFuncVar := "SS1_CPU1215_DO_Vars".DO7.iFuncVar, xOutput => "SS1_CPU1215_DO_Vars".DO7.xInput)
   END_RUNG
   RUNG wire#powerrail
      "DOadv"(xInput := "SS1_CPU1215_DO_Vars".DO7.xInput, xInversion := "SS1_CPU1215_DO_Vars".DO7.xInversion, cMOA := "SS1_CPU1215_DO_Vars".DO7.cMOA, xMemoryOut := "SS1_CPU1215_DO_Vars".DO7.xMemoryOut, xMemoryIn := "SS1_CPU1215_DO_Vars".DO7.xMemoryIn, cMemory := "SS1_CPU1215_DO_Vars".DO7.cMemory, xOutput => "SS1_CPU1215_DO_Vars".DO7.xOutput, iCounterIn := "SS1_CPU1215_DO_Vars".DO7.iCounterIn, iCounterOut := "SS1_CPU1215_DO_Vars".DO7.iCounterOut)
   END_RUNG
   RUNG wire#powerrail
      Contact( "SS1_CPU1215_DO_Vars".DO7.xOutput )
      Coil( "DO11.01.07" )
   END_RUNG
   // the same network as SCL:
   "DOvar"(iFuncSystem := "SS1_CPU1215_DO_Vars".DO7.iFuncSystemID,
           iFuncVar := "SS1_CPU1215_DO_Vars".DO7.iFuncVar,
           xOutput => "SS1_CPU1215_DO_Vars".DO7.xInput);
   "DOadv"(xInput := "SS1_CPU1215_DO_Vars".DO7.xInput,
           xInversion := "SS1_CPU1215_DO_Vars".DO7.xInversion,
           cMOA := "SS1_CPU1215_DO_Vars".DO7.cMOA,
           xMemoryOut := "SS1_CPU1215_DO_Vars".DO7.xMemoryOut,
           xMemoryIn := "SS1_CPU1215_DO_Vars".DO7.xMemoryIn,
           cMemory := "SS1_CPU1215_DO_Vars".DO7.cMemory,
           iCounterIn := "SS1_CPU1215_DO_Vars".DO7.iCounterIn,
           iCounterOut := "SS1_CPU1215_DO_Vars".DO7.iCounterOut,
           xOutput => "SS1_CPU1215_DO_Vars".DO7.xOutput);
   "DO11.01.07" := "SS1_CPU1215_DO_Vars".DO7.xOutput;
END_REGION

REGION Network 26: DQa7
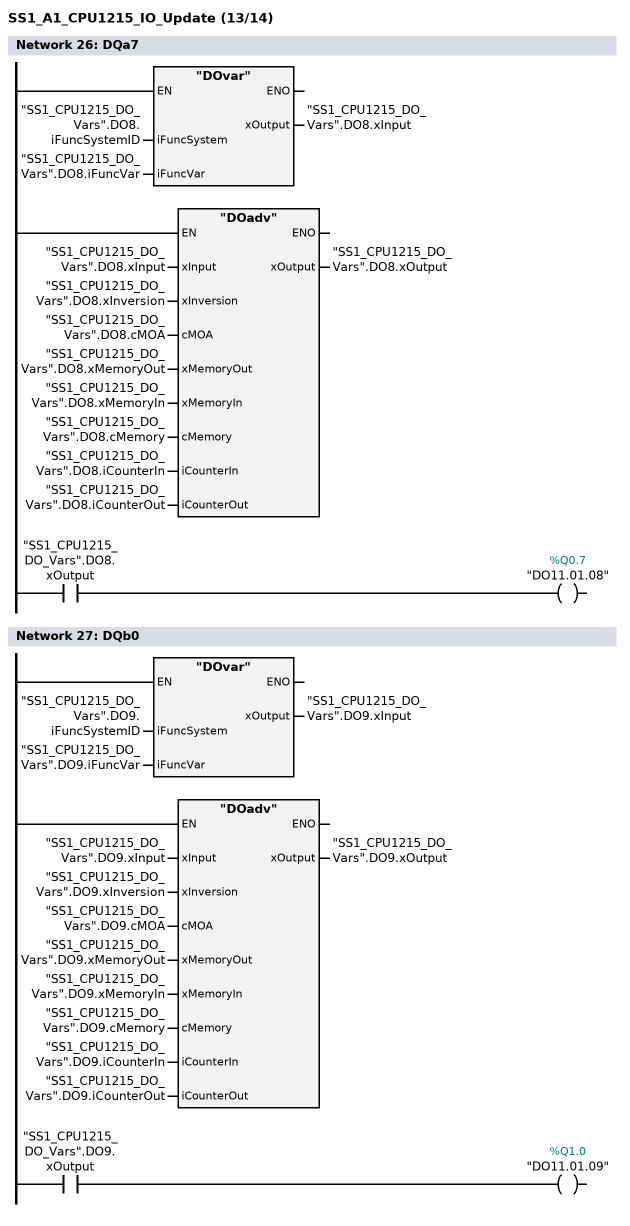
   RUNG wire#powerrail
      "DOvar"(iFuncSystem := "SS1_CPU1215_DO_Vars".DO8.iFuncSystemID, iFuncVar := "SS1_CPU1215_DO_Vars".DO8.iFuncVar, xOutput => "SS1_CPU1215_DO_Vars".DO8.xInput)
   END_RUNG
   RUNG wire#powerrail
      "DOadv"(xInput := "SS1_CPU1215_DO_Vars".DO8.xInput, xInversion := "SS1_CPU1215_DO_Vars".DO8.xInversion, cMOA := "SS1_CPU1215_DO_Vars".DO8.cMOA, xMemoryOut := "SS1_CPU1215_DO_Vars".DO8.xMemoryOut, xMemoryIn := "SS1_CPU1215_DO_Vars".DO8.xMemoryIn, cMemory := "SS1_CPU1215_DO_Vars".DO8.cMemory, xOutput => "SS1_CPU1215_DO_Vars".DO8.xOutput, iCounterIn := "SS1_CPU1215_DO_Vars".DO8.iCounterIn, iCounterOut := "SS1_CPU1215_DO_Vars".DO8.iCounterOut)
   END_RUNG
   RUNG wire#powerrail
      Contact( "SS1_CPU1215_DO_Vars".DO8.xOutput )
      Coil( "DO11.01.08" )
   END_RUNG
   // the same network as SCL:
   "DOvar"(iFuncSystem := "SS1_CPU1215_DO_Vars".DO8.iFuncSystemID,
           iFuncVar := "SS1_CPU1215_DO_Vars".DO8.iFuncVar,
           xOutput => "SS1_CPU1215_DO_Vars".DO8.xInput);
   "DOadv"(xInput := "SS1_CPU1215_DO_Vars".DO8.xInput,
           xInversion := "SS1_CPU1215_DO_Vars".DO8.xInversion,
           cMOA := "SS1_CPU1215_DO_Vars".DO8.cMOA,
           xMemoryOut := "SS1_CPU1215_DO_Vars".DO8.xMemoryOut,
           xMemoryIn := "SS1_CPU1215_DO_Vars".DO8.xMemoryIn,
           cMemory := "SS1_CPU1215_DO_Vars".DO8.cMemory,
           iCounterIn := "SS1_CPU1215_DO_Vars".DO8.iCounterIn,
           iCounterOut := "SS1_CPU1215_DO_Vars".DO8.iCounterOut,
           xOutput => "SS1_CPU1215_DO_Vars".DO8.xOutput);
   "DO11.01.08" := "SS1_CPU1215_DO_Vars".DO8.xOutput;
END_REGION

REGION Network 27: DQb0
   RUNG wire#powerrail
      "DOvar"(iFuncSystem := "SS1_CPU1215_DO_Vars".DO9.iFuncSystemID, iFuncVar := "SS1_CPU1215_DO_Vars".DO9.iFuncVar, xOutput => "SS1_CPU1215_DO_Vars".DO9.xInput)
   END_RUNG
   RUNG wire#powerrail
      "DOadv"(xInput := "SS1_CPU1215_DO_Vars".DO9.xInput, xInversion := "SS1_CPU1215_DO_Vars".DO9.xInversion, cMOA := "SS1_CPU1215_DO_Vars".DO9.cMOA, xMemoryOut := "SS1_CPU1215_DO_Vars".DO9.xMemoryOut, xMemoryIn := "SS1_CPU1215_DO_Vars".DO9.xMemoryIn, cMemory := "SS1_CPU1215_DO_Vars".DO9.cMemory, xOutput => "SS1_CPU1215_DO_Vars".DO9.xOutput, iCounterIn := "SS1_CPU1215_DO_Vars".DO9.iCounterIn, iCounterOut := "SS1_CPU1215_DO_Vars".DO9.iCounterOut)
   END_RUNG
   RUNG wire#powerrail
      Contact( "SS1_CPU1215_DO_Vars".DO9.xOutput )
      Coil( "DO11.01.09" )
   END_RUNG
   // the same network as SCL:
   "DOvar"(iFuncSystem := "SS1_CPU1215_DO_Vars".DO9.iFuncSystemID,
           iFuncVar := "SS1_CPU1215_DO_Vars".DO9.iFuncVar,
           xOutput => "SS1_CPU1215_DO_Vars".DO9.xInput);
   "DOadv"(xInput := "SS1_CPU1215_DO_Vars".DO9.xInput,
           xInversion := "SS1_CPU1215_DO_Vars".DO9.xInversion,
           cMOA := "SS1_CPU1215_DO_Vars".DO9.cMOA,
           xMemoryOut := "SS1_CPU1215_DO_Vars".DO9.xMemoryOut,
           xMemoryIn := "SS1_CPU1215_DO_Vars".DO9.xMemoryIn,
           cMemory := "SS1_CPU1215_DO_Vars".DO9.cMemory,
           iCounterIn := "SS1_CPU1215_DO_Vars".DO9.iCounterIn,
           iCounterOut := "SS1_CPU1215_DO_Vars".DO9.iCounterOut,
           xOutput => "SS1_CPU1215_DO_Vars".DO9.xOutput);
   "DO11.01.09" := "SS1_CPU1215_DO_Vars".DO9.xOutput;
END_REGION

REGION Network 28: DQb1
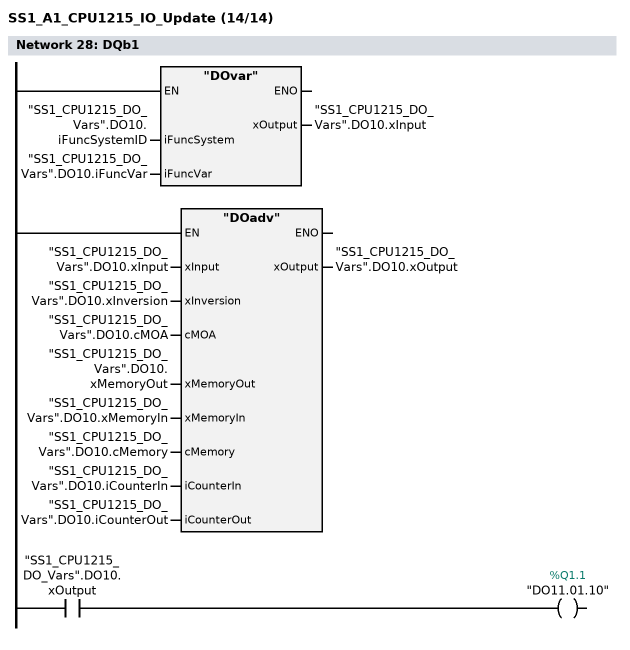
   RUNG wire#powerrail
      "DOvar"(iFuncSystem := "SS1_CPU1215_DO_Vars".DO10.iFuncSystemID, iFuncVar := "SS1_CPU1215_DO_Vars".DO10.iFuncVar, xOutput => "SS1_CPU1215_DO_Vars".DO10.xInput)
   END_RUNG
   RUNG wire#powerrail
      "DOadv"(xInput := "SS1_CPU1215_DO_Vars".DO10.xInput, xInversion := "SS1_CPU1215_DO_Vars".DO10.xInversion, cMOA := "SS1_CPU1215_DO_Vars".DO10.cMOA, xMemoryOut := "SS1_CPU1215_DO_Vars".DO10.xMemoryOut, xMemoryIn := "SS1_CPU1215_DO_Vars".DO10.xMemoryIn, cMemory := "SS1_CPU1215_DO_Vars".DO10.cMemory, xOutput => "SS1_CPU1215_DO_Vars".DO10.xOutput, iCounterIn := "SS1_CPU1215_DO_Vars".DO10.iCounterIn, iCounterOut := "SS1_CPU1215_DO_Vars".DO10.iCounterOut)
   END_RUNG
   RUNG wire#powerrail
      Contact( "SS1_CPU1215_DO_Vars".DO10.xOutput )
      Coil( "DO11.01.10" )
   END_RUNG
   // the same network as SCL:
   "DOvar"(iFuncSystem := "SS1_CPU1215_DO_Vars".DO10.iFuncSystemID,
           iFuncVar := "SS1_CPU1215_DO_Vars".DO10.iFuncVar,
           xOutput => "SS1_CPU1215_DO_Vars".DO10.xInput);
   "DOadv"(xInput := "SS1_CPU1215_DO_Vars".DO10.xInput,
           xInversion := "SS1_CPU1215_DO_Vars".DO10.xInversion,
           cMOA := "SS1_CPU1215_DO_Vars".DO10.cMOA,
           xMemoryOut := "SS1_CPU1215_DO_Vars".DO10.xMemoryOut,
           xMemoryIn := "SS1_CPU1215_DO_Vars".DO10.xMemoryIn,
           cMemory := "SS1_CPU1215_DO_Vars".DO10.cMemory,
           iCounterIn := "SS1_CPU1215_DO_Vars".DO10.iCounterIn,
           iCounterOut := "SS1_CPU1215_DO_Vars".DO10.iCounterOut,
           xOutput => "SS1_CPU1215_DO_Vars".DO10.xOutput);
   "DO11.01.10" := "SS1_CPU1215_DO_Vars".DO10.xOutput;
END_REGION
END_FUNCTION

FUNCTION "AIvars" : Void   // FC10014, LAD
{ S7_Optimized_Access := 'TRUE' }
VERSION : 0.1
// stored: AutoNumber false, IsIECCheckEnabled false, SetENOAutomatically false, UDAEnableTagReadback false
   VAR_INPUT
      rInput : Real;
      iFuncSystem : Byte;
      iFuncVar : Byte;
   END_VAR
BEGIN

REGION Network 1 (SCL)
   CASE #iFuncSystem OF
       0:  // Statement section case 2 to 4
           ;
       1..3:  // Statement section case 1
           CASE #iFuncVar OF
               0:  //
                   ;
               1:  //
                   "AHUAI".AI.rIAQ[#iFuncSystem] := #rInput;
               2:  // 
                   "AHUAI".AI.rBuildingdP[#iFuncSystem] := #rInput;
               3:  // 
                   "AHUAI".AI.rRoomAirTemp_PLC_AI[#iFuncSystem] := #rInput;
               4:  // 
                   "AHUAI".AI.rSupplyAirTemp[#iFuncSystem] := #rInput;
               5:  // 
                   "AHUAI".AI.rReturnAirTemp[#iFuncSystem] := #rInput;
               6:  // 
                   "AHUAI".AI.rFrostProtWaterTemp[#iFuncSystem] := #rInput;
               7:  // 
                   "AHUAI".AI.rFrostProtAirTemp[#iFuncSystem] := #rInput;
               8:  // 
                   "AHUAI".AI.rRoomAirRelHumi[#iFuncSystem] := #rInput;
               9:  // reserve
                   "AHUAI".AI.rReserve[#iFuncSystem] := #rInput;;
               10:  // 
                   "AHUAI".AI.rSAFilterdP[#iFuncSystem] := #rInput;
               11:
                   "AHUAI".AI.rSAFFlow[#iFuncSystem] := #rInput;
               12:
                   "AHUAI".AI.rRoomAirTemp_Actual[#iFuncSystem] := #rInput;
               13:
                   "AHUAI".AI.rRoomAirTemp_LoraAvg[#iFuncSystem] := #rInput;
               14:
                   "AHUAI".AI.rRoomAirTemp_MSensor[#iFuncSystem] := #rInput;
               ELSE
                   ;
           END_CASE;
       4..9:
           ;
       10:
           CASE #iFuncVar OF
               0:  // 
                   ;
               1:  // 
                   "HSsAI".AI.rHSBoilerRoomTemp := #rInput;
               2:  // 
                   "HSsAI".AI.rHSWaterPressure := #rInput;
               3:  // 
                   "HSsAI".AI.rHSSupplyMainfoldTemp := #rInput;
               4:  // 
                   "HSsAI".AI.rOutdoorTemp_PLC_AI := #rInput;
               5:    
                   "HCsAI".AI.rSupplyWaterTemp[1] := #rInput;
               6:  // 
                   "HCsAI".AI.rReturnWaterTemp[1] := #rInput;
               7:  // 
                   "HCsAI".AI.r3vwPosFbk[1] := #rInput;
               8:    
                   "HCsAI".AI.rSupplyWaterTemp[2] := #rInput;
               9:  // 
                   "HCsAI".AI.rReturnWaterTemp[2] := #rInput;
               10:  // 
                   "HCsAI".AI.r3vwPosFbk[2] := #rInput;
               ELSE
                   ;
           END_CASE;
       11..13:
           ;
       14:
           CASE #iFuncVar OF
               0:  // 
                   ;
               1:
                   "DHWAI".AI.r14200a := #rInput;
               2:  // 
                   "DHWAI".AI.r14201a := #rInput;
               ELSE
                   ;
           END_CASE;
       15..20:
           ;
       21: //Proxy Channels    
           CASE #iFuncVar OF
               0:  //
                   ;
               1..8:  //
                   "AHUProxyCH".Vars.rCHDrivenSignal[#iFuncVar] := #rInput;
               ELSE
                   ;
           END_CASE;
       22..99:
           ;
       100: //Diesel Line   
           CASE #iFuncVar OF
               0:  //
                   ;
               1:  //
                   "DLsAI".AI.rDayTankLevel[1] := #rInput;
               2:  //
                   "DLsAI".AI.rDayTankLevel[2] := #rInput;
               ELSE
                   ;
           END_CASE;
       ELSE  // Statement section ELSE
           ;
   END_CASE;
END_REGION
END_FUNCTION

FUNCTION "AOvar" : Void   // FC10011, LAD
{ S7_Optimized_Access := 'TRUE' }
VERSION : 0.1
// stored: AutoNumber false, IsIECCheckEnabled false, SetENOAutomatically false, UDAEnableTagReadback false
   VAR_INPUT
      iFuncSystem : Byte;
      iFuncVar : Byte;
   END_VAR
   VAR_OUTPUT
      rOutput : Real;
   END_VAR
BEGIN

REGION Network 1 (SCL)
   CASE #iFuncSystem OF
       0:  // Statement section case 2 to 4
           ;
       1..3:  // Statement section case 1
           CASE #iFuncVar OF
               0:  // 
                   ;
               1:  // 
                   #rOutput := "AHUAO".AO.rSAFAnalog[#iFuncSystem];
               2:  // 
                   #rOutput := "AHUAO".AO.rHeater[#iFuncSystem];
               3:  // 
                   #rOutput := "AHUAO".AO.rMixingAirDumper[#iFuncSystem];
               4:  // 
                   #rOutput := "AHUAO".AO.rExtractAirDumper[#iFuncSystem];
               5:  // 
                   #rOutput := "AHUAO".AO.rCooler[#iFuncSystem];
               6:  // 
                   #rOutput := "AHUAO".AO.rWHU[#iFuncSystem];
           END_CASE;
       4..20:
           ;
       21: //Proxy Channels    
           CASE #iFuncVar OF
               0:  //
                   ;
               1..8:  //
                   #rOutput := "AHUProxyCH".Vars.rCHProxySignal[#iFuncVar];
               ELSE
                   ;
           END_CASE;
       ELSE  // Statement section ELSE
           ;
   END_CASE;
END_REGION
END_FUNCTION

FUNCTION "AOadv" : Void   // FC10012, FBD
{ S7_Optimized_Access := 'TRUE' }
VERSION : 0.1
// stored: AutoNumber false, IsIECCheckEnabled false, SetENOAutomatically false, UDAEnableTagReadback false
   VAR_INPUT
      rInput : Real;   // 0 to 100
      cM0A : Byte;   // 0-direct / 1-reverse / 0-outp_off / 1- out=MAN_OUTPUT /2 -out=input
      rManOutput : Real;
   END_VAR
   VAR_OUTPUT
      iOutput : Int;
   END_VAR
   VAR_TEMP
      rOut : Real;
      rOutScaled : Real;
      rManOutputTemp : Real;
      iManOutputTemp : Int;
   END_VAR
   VAR CONSTANT
      iRawMin : Int := 0;
      iRawMax : Int := 27648;
   END_VAR
BEGIN

REGION Network 1 (SCL): // --- Вибір режиму ---
   // --- Вибір режиму ---
   CASE #cM0A OF
       0: // Off
           #rOut := 0.0;
       1: // Manual
           #rOut := #rManOutput;
       2: // Auto
           #rOut := #rInput;
       ELSE
           #rOut := 0.0; // захист від некоректних значень
   END_CASE;
END_REGION

REGION Network 2 (SCL): // --- Обмеження в межах 0.0…100.0 ---
   // --- Обмеження в межах 0.0…100.0 ---
   IF #rOut < 0.0 THEN
       #rOut := 0.0;
   ELSIF
       #rOut > 100.0 THEN
       #rOut := 100.0;
   END_IF;
END_REGION

REGION Network 3 (SCL)
   #rOutScaled := (#rOut * 27648.0) / 100;
END_REGION

REGION Network 4 (SCL)
   IF #rOutScaled < 0.0 THEN
       #rOutScaled := 0.0;
   ELSIF
       #rOutScaled > 27648.0 THEN
       #rOutScaled := 27648.0;
   END_IF;
END_REGION

REGION Network 5 (SCL)
   #iOutput := REAL_TO_INT(#rOutScaled + 0.5);
END_REGION
END_FUNCTION

FUNCTION "DIvars" : Void   // FC10008, LAD
{ S7_Optimized_Access := 'TRUE' }
VERSION : 0.1
// stored: AutoNumber false, IsIECCheckEnabled false, SetENOAutomatically false, UDAEnableTagReadback false
   VAR_INPUT
      xInput : Bool;
      iFuncSystem : Byte;
      iFuncVar : Byte;
   END_VAR
BEGIN

REGION Network 1 (SCL)
   CASE #iFuncSystem OF
       0:  // Statement section case 2 to 4
           ;
       1..3:  // Statement section case 1
           CASE #iFuncVar OF
               0:  // 
                   ;
               1:  // 
                   "AHUDI".DI.xHeaterPumpReady[#iFuncSystem] := #xInput;
               2:  // 
                   "AHUDI".DI.xHeaterPumpInd[#iFuncSystem] := #xInput;
               3:  // 
                   "AHUDI".DI.xHeaterPumpAlarm[#iFuncSystem] := #xInput;
               4:  // 
                   "AHUDI".DI.xSAFAnalogReady[#iFuncSystem] := #xInput;
               5:  // 
                   "AHUDI".DI.xSAFAnalogInd[#iFuncSystem] := #xInput;
               6:  // 
                   "AHUDI".DI.xSAFAnalogAlarm[#iFuncSystem] := #xInput;
               7:  // 
                   "AHUDI".DI.xSAFSp1Ready[#iFuncSystem] := #xInput;
               8:  // 
                   "AHUDI".DI.xSAFSp1Ind[#iFuncSystem] := #xInput;
               9:  // 
                   "AHUDI".DI.xSAFSp1Alarm[#iFuncSystem] := #xInput;
               10:  // 
                   "AHUDI".DI.xSAFSp2Ready[#iFuncSystem] := #xInput;
               11:  // 
                   "AHUDI".DI.xSAFSp2Ind[#iFuncSystem] := #xInput;
               12:  // 
                   "AHUDI".DI.xSAFSp2Alarm[#iFuncSystem] := #xInput;
               13:  // 
                   "AHUDI".DI.xSAFdPInd[#iFuncSystem] := #xInput;
               14:  // 
                   "AHUDI".DI.xFrostProtTstat[#iFuncSystem] := #xInput;
               15:  // 
                   "AHUDI".DI.xSAFdPAlarm[#iFuncSystem] := #xInput;
               16:  // 
                   "AHUDI".DI.xSAFPanelSelectorOff[#iFuncSystem] := #xInput;
               17:  // 
                   "AHUDI".DI.xSAFPanelSelector1St[#iFuncSystem] := #xInput;
               18:  // 
                   "AHUDI".DI.xSAFPanelSelector2St[#iFuncSystem] := #xInput;
               19:  // 
                   "AHUDI".DI.xSAFPanelSelectorAuto[#iFuncSystem] := #xInput;
               20:  //
                   "AHUDI".DI.xSAFMotorPTCAlarm[#iFuncSystem] := #xInput;
               21:  //
                   "AHUDI".DI.xReserve1[#iFuncSystem] := #xInput;
               ELSE
                   ;
           END_CASE;
       4..9:
           ;
       10:  //    
           CASE #iFuncVar OF
               0:  //
                   ;
               1:
                   "HCsDI".Requests.xHCPump1Ready[1] := #xInput;
               2:
                   "HCsDI".Requests.xHCPump1Ind[1] := #xInput;
               3: //    
                   "HCsDI".Requests.xHCPump1Alarm[1] := #xInput;
               4:  //
                   "HCsDI".Requests.xHCPump2Ready[1] := #xInput;
               5:  //
                   "HCsDI".Requests.xHCPump2Ind[1] := #xInput;
               6:  //
                   "HCsDI".Requests.xHCPump2Alarm[1] := #xInput;
               7:  //
                   "HCsDI".Requests.xHCDoublePumpInAuto[1] := #xInput;
               8:
                   "HCsDI".Requests.xHCPump1Ready[2] := #xInput;
               9:
                   "HCsDI".Requests.xHCPump1Ind[2] := #xInput;
               10: //    
                   "HCsDI".Requests.xHCPump1Alarm[2] := #xInput;
               11:  //
                   "HCsDI".Requests.xHCPump2Ready[2] := #xInput;
               12:  //
                   "HCsDI".Requests.xHCPump2Ind[2] := #xInput;
               13:  //
                   "HCsDI".Requests.xHCPump2Alarm[2] := #xInput;
               14:  //
                   "HCsDI".Requests.xHCDoublePumpInAuto[2] := #xInput;
               15..20: //
                   ;
               21:  //
                   "HSsDI".Requests.xBoilerShuntPumpReady[1] := #xInput;
               22:  //
                   "HSsDI".Requests.xBoilerShuntPumpInd[1] := #xInput;
               23:  //
                   "HSsDI".Requests.xBoilerShuntPumpAlarm[1] := #xInput;
               24:  //
                   "HSsDI".Requests.xBoilerShuntPumpInAuto[1] := #xInput;
               25:  //
                   "HSsDI".Requests.xBoilerStage1Ind[1] := #xInput;
               26:  //
                   "HSsDI".Requests.xBoilerStage2Ind[1] := #xInput;
               27:  //
                   "HSsDI".Requests.xBurnerAlarm[1] := #xInput;
               28:  //
                   "HSsDI".Requests.xBoilerAlarm[1] := #xInput;
               29:  //
                   "HSsDI".Requests.xBoilerReady[1] := #xInput;
               30:  //
                   "HSsDI".Requests.xBoilerReserve[1] := #xInput;
               31:  //
                   "HSsDI".Requests.xBoilerShuntPumpReady[2] := #xInput;
               32:  //
                   "HSsDI".Requests.xBoilerShuntPumpInd[2] := #xInput;
               33:  //
                   "HSsDI".Requests.xBoilerShuntPumpAlarm[2] := #xInput;
               34:  //
                   "HSsDI".Requests.xBoilerShuntPumpInAuto[2] := #xInput;
               35:  //
                   "HSsDI".Requests.xBoilerStage1Ind[2] := #xInput;
               36:  //
                   "HSsDI".Requests.xBoilerStage2Ind[2] := #xInput;
               37:  //
                   "HSsDI".Requests.xBurnerAlarm[2] := #xInput;
               38:  //
                   "HSsDI".Requests.xBoilerAlarm[2] := #xInput;
               39:  //
                   "HSsDI".Requests.xBoilerReady[2] := #xInput;
               40:  //
                   "HSsDI".Requests.xBoilerReserve[2] := #xInput;
               41:
                   "HSsDI".Requests.xSeasonWinter[1] := #xInput;
               42:
                   "HSsDI".Requests.xSeasonSummer[1] := #xInput;
               43:
                   "HSsDI".Requests.xSeasonAuto[1] := #xInput;
               44:
                   "HSsDI".Requests.xSeasonWinter[2] := #xInput;
               45:
                   "HSsDI".Requests.xSeasonSummer[2] := #xInput;
               46:
                   "HSsDI".Requests.xSeasonAuto[2] := #xInput;
               ELSE
                   ;
           END_CASE;
       11..20:
           ;
       21:
           CASE #iFuncVar OF
           0:
               ;
           1..8:
               "AHUProxyCH".Vars.xCHRlyIsOnInd[#iFuncVar] := #xInput;
           9..16:
               "AHUProxyCH".Vars.xCHRlyIsOffInd[#iFuncVar] := #xInput;
           ELSE
               ;
           END_CASE;
       22..99:
           ;
       100:
           CASE #iFuncVar OF
               0:
                   ;
               1:
                   "DLsDI".Requests.xDieselLineHeatingReady[1] := #xInput;
               2:
                   "DLsDI".Requests.xDieselLineHeatingReady[2] := #xInput;
               3:
                   "DLsDI".Requests.xDieselLineHeatingInd[1]:= #xInput;
               4:
                   "DLsDI".Requests.xDieselLineHeatingInd[2] := #xInput;
               5:
                   "DLsDI".Requests.xDieselLinePumpInd[1] := #xInput;
               6:
                   "DLsDI".Requests.xDieselLinePumpInd[2]:= #xInput;
               7:
                   "DLsDI".Requests.xDieselLinePnom := #xInput;
               8:
                   "DLsDI".Requests.xDieselLineValveToBoilerInd := #xInput;
               9:
                   "DLsDI".Requests.xDieselLinePmax:= #xInput;
               10:
                   "DLsDI".Requests.xDieselLinePumpZoneWaterFloodAlarm := #xInput;
               11:
                   "DLsDI".Requests.xDieselLineMainTankDoubleWallAlarmInd := #xInput;
               12:
                   "DLsDI".Requests.xDieselLineMainTankMinLevelInd:= #xInput;
               13:
                   "DLsDI".Requests.Reserve1 := #xInput;
               14:
                   "DLsDI".Requests.Reserve2 := #xInput;
               15:
                   "DLsDI".Requests.xDieselLinePumpPanelSelectorOff:= #xInput;
               16:
                   "DLsDI".Requests.xDieselLinePumpPanelSelectorP1Man := #xInput;
               17:
                   "DLsDI".Requests.xDieselLinePumpPanelSelectorP2Man := #xInput;
               18:
                   "DLsDI".Requests.xDieselLinePumpPanelSelectorAuto:= #xInput;
               ELSE
                   ;
           END_CASE;
       ELSE  // Statement section ELSE
           ;
   END_CASE;
END_REGION
END_FUNCTION

FUNCTION "DOvar" : Void   // FC10010, LAD
{ S7_Optimized_Access := 'TRUE' }
VERSION : 0.1
// stored: AutoNumber false, IsIECCheckEnabled false, SetENOAutomatically false, UDAEnableTagReadback false
   VAR_INPUT
      iFuncSystem : Byte;
      iFuncVar : Byte;
   END_VAR
   VAR_OUTPUT
      xOutput : Bool;
   END_VAR
BEGIN

REGION Network 1 (SCL)
   CASE #iFuncSystem OF
       0:  // Statement section case 2 to 4
           ;
       1..3:  // Statement section case 1
           CASE #iFuncVar OF
               0:  // 
                   ;
               1:  // 
                   #xOutput := "AHUDO".Requests.xHeaterPumpCmd[#iFuncSystem];
               2:  // 
                   #xOutput := "AHUDO".Requests.xSAFAnalogEnable[#iFuncSystem];
               3:  // 
                   #xOutput := "AHUDO".Requests.xSAFSp1Cmd[#iFuncSystem];
               4:  // 
                   #xOutput := "AHUDO".Requests.xSAFSp2Cmd[#iFuncSystem];
           END_CASE;
        4..9:
            ;
        10:
            CASE #iFuncVar OF
                0:  // 
                    ;
                1:  // 
                    #xOutput := "HCsDO".Requests.xHC3wvIncrease[1];
                2:  // 
                    #xOutput := "HCsDO".Requests.xHC3wvDecrease[1];
                3:  // 
                    #xOutput := "HCsDO".Requests.xHC3wvIncrease[2];
                4:  // 
                    #xOutput := "HCsDO".Requests.xHC3wvDecrease[2];
                5:  //
                    #xOutput := "HCsDO".Requests.xHCPump1Cmd[1];
                6:  //
                    #xOutput := "HCsDO".Requests.xHCPump2Cmd[1];
                7:  //
                    #xOutput := "HCsDO".Requests.xHCPump1Cmd[2];
                8:  //
                    #xOutput := "HCsDO".Requests.xHCPump2Cmd[2];
                9:  //    
                    ;
                10:
                    #xOutput := "HSsDO".Requests.xBoilerEnable[1];
                11:
                    #xOutput := "HSsDO".Requests.xBoilerSt1Enable[1];
                12:
                    #xOutput := "HSsDO".Requests.xBoilerSt2Enable[1];
                13:
                    #xOutput := "HSsDO".Requests.xBoilerShuntPumpEnable[1];
                14:
                    #xOutput := "HSsDO".Requests.xBoilerShutOffValveCmd[1];
                15:
                    ;
                16:
                    #xOutput := "HSsDO".Requests.xBoilerEnable[2];
                17:
                    #xOutput := "HSsDO".Requests.xBoilerSt1Enable[2];
                18:
                    #xOutput := "HSsDO".Requests.xBoilerSt2Enable[2];
                19:
                    #xOutput := "HSsDO".Requests.xBoilerShuntPumpEnable[2];
                20:
                    #xOutput := "HSsDO".Requests.xBoilerShutOffValveCmd[2];
                ELSE:
                    ;
            END_CASE;
        11..99:
            ;
        100:    //DieselLine
            CASE #iFuncVar OF
                0:  // 
                    ;
                1:  // 
                    #xOutput := "DLsDO".Requests.xDieselLineHeatingCmd[1];
                2:  // 
                    #xOutput := "DLsDO".Requests.xDieselLineHeatingCmd[2];
                3:  // 
                    #xOutput := "DLsDO".Requests.xDieselLinePumpEnable;
                4:  // 
                    #xOutput := "DLsDO".Requests.xDieselLinePumpSelect;
                5:  //
                    #xOutput := "DLsDO".Requests.xDieselLineDayTankValve[1];
                6:  //
                    #xOutput := "DLsDO".Requests.xDieselLineDayTankValve[2];
                ELSE:
                    ;
            END_CASE;
       ELSE  // Statement section ELSE
           ;
   END_CASE;
END_REGION
END_FUNCTION

FUNCTION "HeatingPLC_vIO" : Void   // FC11001, LAD
{ S7_Optimized_Access := 'FALSE' }
VERSION : 0.1
// stored: AutoNumber false, IsIECCheckEnabled false, SetENOAutomatically false, UDAEnableTagReadback false
BEGIN

REGION Network 1
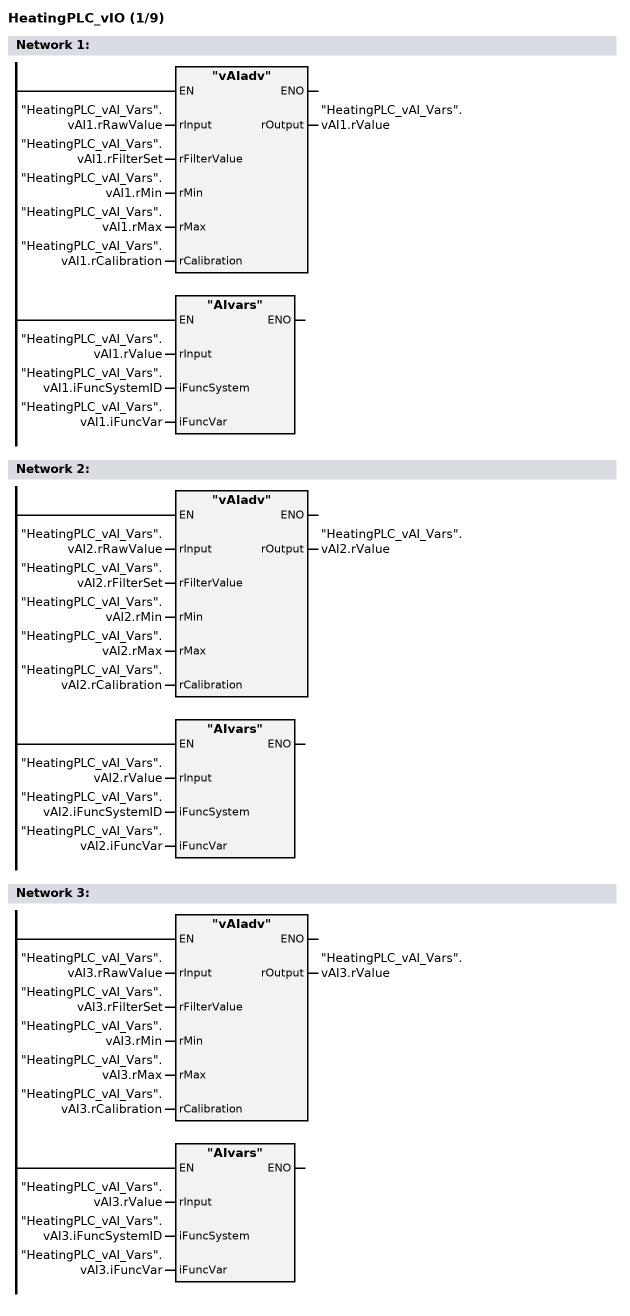
   RUNG wire#powerrail
      "vAIadv"(rInput := "HeatingPLC_vAI_Vars".vAI1.rRawValue, rFilterValue := "HeatingPLC_vAI_Vars".vAI1.rFilterSet, rMin := "HeatingPLC_vAI_Vars".vAI1.rMin, rMax := "HeatingPLC_vAI_Vars".vAI1.rMax, rCalibration := "HeatingPLC_vAI_Vars".vAI1.rCalibration, rOutput => "HeatingPLC_vAI_Vars".vAI1.rValue)
   END_RUNG
   RUNG wire#powerrail
      "AIvars"(rInput := "HeatingPLC_vAI_Vars".vAI1.rValue, iFuncSystem := "HeatingPLC_vAI_Vars".vAI1.iFuncSystemID, iFuncVar := "HeatingPLC_vAI_Vars".vAI1.iFuncVar)
   END_RUNG
   // the same network as SCL:
   "vAIadv"(rInput := "HeatingPLC_vAI_Vars".vAI1.rRawValue,
            rFilterValue := "HeatingPLC_vAI_Vars".vAI1.rFilterSet,
            rMin := "HeatingPLC_vAI_Vars".vAI1.rMin,
            rMax := "HeatingPLC_vAI_Vars".vAI1.rMax,
            rCalibration := "HeatingPLC_vAI_Vars".vAI1.rCalibration,
            rOutput => "HeatingPLC_vAI_Vars".vAI1.rValue);
   "AIvars"(rInput := "HeatingPLC_vAI_Vars".vAI1.rValue,
            iFuncSystem := "HeatingPLC_vAI_Vars".vAI1.iFuncSystemID,
            iFuncVar := "HeatingPLC_vAI_Vars".vAI1.iFuncVar);
END_REGION

REGION Network 2
   RUNG wire#powerrail
      "vAIadv"(rInput := "HeatingPLC_vAI_Vars".vAI2.rRawValue, rFilterValue := "HeatingPLC_vAI_Vars".vAI2.rFilterSet, rMin := "HeatingPLC_vAI_Vars".vAI2.rMin, rMax := "HeatingPLC_vAI_Vars".vAI2.rMax, rCalibration := "HeatingPLC_vAI_Vars".vAI2.rCalibration, rOutput => "HeatingPLC_vAI_Vars".vAI2.rValue)
   END_RUNG
   RUNG wire#powerrail
      "AIvars"(rInput := "HeatingPLC_vAI_Vars".vAI2.rValue, iFuncSystem := "HeatingPLC_vAI_Vars".vAI2.iFuncSystemID, iFuncVar := "HeatingPLC_vAI_Vars".vAI2.iFuncVar)
   END_RUNG
   // the same network as SCL:
   "vAIadv"(rInput := "HeatingPLC_vAI_Vars".vAI2.rRawValue,
            rFilterValue := "HeatingPLC_vAI_Vars".vAI2.rFilterSet,
            rMin := "HeatingPLC_vAI_Vars".vAI2.rMin,
            rMax := "HeatingPLC_vAI_Vars".vAI2.rMax,
            rCalibration := "HeatingPLC_vAI_Vars".vAI2.rCalibration,
            rOutput => "HeatingPLC_vAI_Vars".vAI2.rValue);
   "AIvars"(rInput := "HeatingPLC_vAI_Vars".vAI2.rValue,
            iFuncSystem := "HeatingPLC_vAI_Vars".vAI2.iFuncSystemID,
            iFuncVar := "HeatingPLC_vAI_Vars".vAI2.iFuncVar);
END_REGION

REGION Network 3
   RUNG wire#powerrail
      "vAIadv"(rInput := "HeatingPLC_vAI_Vars".vAI3.rRawValue, rFilterValue := "HeatingPLC_vAI_Vars".vAI3.rFilterSet, rMin := "HeatingPLC_vAI_Vars".vAI3.rMin, rMax := "HeatingPLC_vAI_Vars".vAI3.rMax, rCalibration := "HeatingPLC_vAI_Vars".vAI3.rCalibration, rOutput => "HeatingPLC_vAI_Vars".vAI3.rValue)
   END_RUNG
   RUNG wire#powerrail
      "AIvars"(rInput := "HeatingPLC_vAI_Vars".vAI3.rValue, iFuncSystem := "HeatingPLC_vAI_Vars".vAI3.iFuncSystemID, iFuncVar := "HeatingPLC_vAI_Vars".vAI3.iFuncVar)
   END_RUNG
   // the same network as SCL:
   "vAIadv"(rInput := "HeatingPLC_vAI_Vars".vAI3.rRawValue,
            rFilterValue := "HeatingPLC_vAI_Vars".vAI3.rFilterSet,
            rMin := "HeatingPLC_vAI_Vars".vAI3.rMin,
            rMax := "HeatingPLC_vAI_Vars".vAI3.rMax,
            rCalibration := "HeatingPLC_vAI_Vars".vAI3.rCalibration,
            rOutput => "HeatingPLC_vAI_Vars".vAI3.rValue);
   "AIvars"(rInput := "HeatingPLC_vAI_Vars".vAI3.rValue,
            iFuncSystem := "HeatingPLC_vAI_Vars".vAI3.iFuncSystemID,
            iFuncVar := "HeatingPLC_vAI_Vars".vAI3.iFuncVar);
END_REGION

REGION Network 4
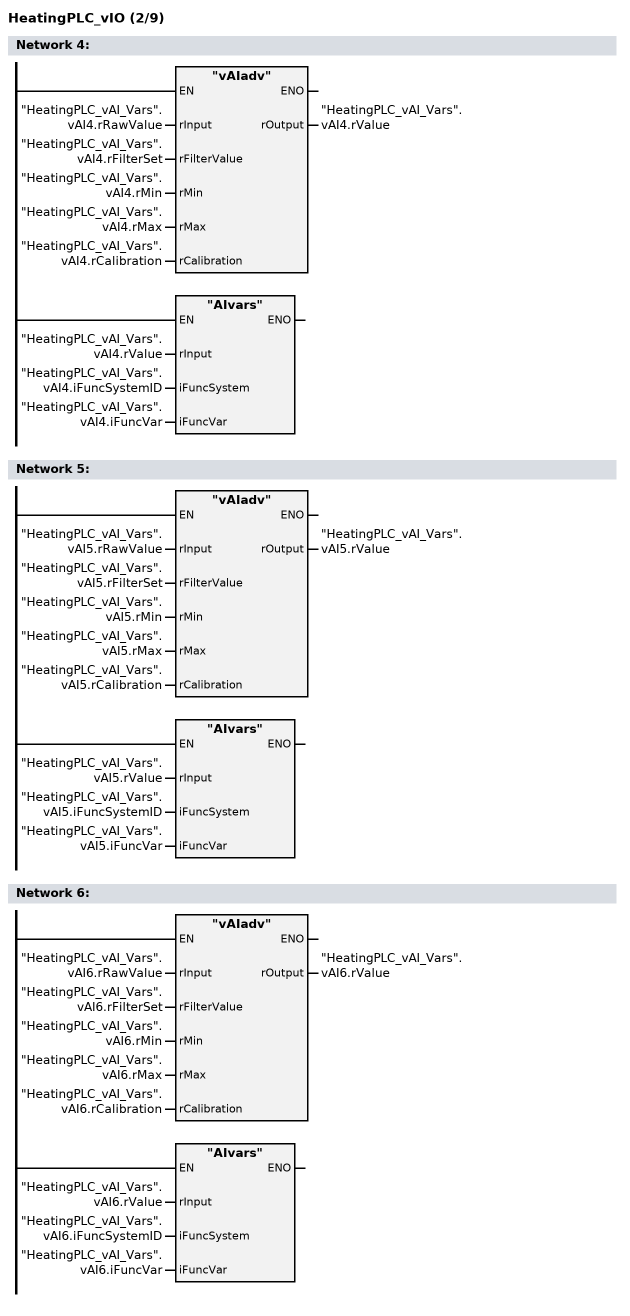
   RUNG wire#powerrail
      "vAIadv"(rInput := "HeatingPLC_vAI_Vars".vAI4.rRawValue, rFilterValue := "HeatingPLC_vAI_Vars".vAI4.rFilterSet, rMin := "HeatingPLC_vAI_Vars".vAI4.rMin, rMax := "HeatingPLC_vAI_Vars".vAI4.rMax, rCalibration := "HeatingPLC_vAI_Vars".vAI4.rCalibration, rOutput => "HeatingPLC_vAI_Vars".vAI4.rValue)
   END_RUNG
   RUNG wire#powerrail
      "AIvars"(rInput := "HeatingPLC_vAI_Vars".vAI4.rValue, iFuncSystem := "HeatingPLC_vAI_Vars".vAI4.iFuncSystemID, iFuncVar := "HeatingPLC_vAI_Vars".vAI4.iFuncVar)
   END_RUNG
   // the same network as SCL:
   "vAIadv"(rInput := "HeatingPLC_vAI_Vars".vAI4.rRawValue,
            rFilterValue := "HeatingPLC_vAI_Vars".vAI4.rFilterSet,
            rMin := "HeatingPLC_vAI_Vars".vAI4.rMin,
            rMax := "HeatingPLC_vAI_Vars".vAI4.rMax,
            rCalibration := "HeatingPLC_vAI_Vars".vAI4.rCalibration,
            rOutput => "HeatingPLC_vAI_Vars".vAI4.rValue);
   "AIvars"(rInput := "HeatingPLC_vAI_Vars".vAI4.rValue,
            iFuncSystem := "HeatingPLC_vAI_Vars".vAI4.iFuncSystemID,
            iFuncVar := "HeatingPLC_vAI_Vars".vAI4.iFuncVar);
END_REGION

REGION Network 5
   RUNG wire#powerrail
      "vAIadv"(rInput := "HeatingPLC_vAI_Vars".vAI5.rRawValue, rFilterValue := "HeatingPLC_vAI_Vars".vAI5.rFilterSet, rMin := "HeatingPLC_vAI_Vars".vAI5.rMin, rMax := "HeatingPLC_vAI_Vars".vAI5.rMax, rCalibration := "HeatingPLC_vAI_Vars".vAI5.rCalibration, rOutput => "HeatingPLC_vAI_Vars".vAI5.rValue)
   END_RUNG
   RUNG wire#powerrail
      "AIvars"(rInput := "HeatingPLC_vAI_Vars".vAI5.rValue, iFuncSystem := "HeatingPLC_vAI_Vars".vAI5.iFuncSystemID, iFuncVar := "HeatingPLC_vAI_Vars".vAI5.iFuncVar)
   END_RUNG
   // the same network as SCL:
   "vAIadv"(rInput := "HeatingPLC_vAI_Vars".vAI5.rRawValue,
            rFilterValue := "HeatingPLC_vAI_Vars".vAI5.rFilterSet,
            rMin := "HeatingPLC_vAI_Vars".vAI5.rMin,
            rMax := "HeatingPLC_vAI_Vars".vAI5.rMax,
            rCalibration := "HeatingPLC_vAI_Vars".vAI5.rCalibration,
            rOutput => "HeatingPLC_vAI_Vars".vAI5.rValue);
   "AIvars"(rInput := "HeatingPLC_vAI_Vars".vAI5.rValue,
            iFuncSystem := "HeatingPLC_vAI_Vars".vAI5.iFuncSystemID,
            iFuncVar := "HeatingPLC_vAI_Vars".vAI5.iFuncVar);
END_REGION

REGION Network 6
   RUNG wire#powerrail
      "vAIadv"(rInput := "HeatingPLC_vAI_Vars".vAI6.rRawValue, rFilterValue := "HeatingPLC_vAI_Vars".vAI6.rFilterSet, rMin := "HeatingPLC_vAI_Vars".vAI6.rMin, rMax := "HeatingPLC_vAI_Vars".vAI6.rMax, rCalibration := "HeatingPLC_vAI_Vars".vAI6.rCalibration, rOutput => "HeatingPLC_vAI_Vars".vAI6.rValue)
   END_RUNG
   RUNG wire#powerrail
      "AIvars"(rInput := "HeatingPLC_vAI_Vars".vAI6.rValue, iFuncSystem := "HeatingPLC_vAI_Vars".vAI6.iFuncSystemID, iFuncVar := "HeatingPLC_vAI_Vars".vAI6.iFuncVar)
   END_RUNG
   // the same network as SCL:
   "vAIadv"(rInput := "HeatingPLC_vAI_Vars".vAI6.rRawValue,
            rFilterValue := "HeatingPLC_vAI_Vars".vAI6.rFilterSet,
            rMin := "HeatingPLC_vAI_Vars".vAI6.rMin,
            rMax := "HeatingPLC_vAI_Vars".vAI6.rMax,
            rCalibration := "HeatingPLC_vAI_Vars".vAI6.rCalibration,
            rOutput => "HeatingPLC_vAI_Vars".vAI6.rValue);
   "AIvars"(rInput := "HeatingPLC_vAI_Vars".vAI6.rValue,
            iFuncSystem := "HeatingPLC_vAI_Vars".vAI6.iFuncSystemID,
            iFuncVar := "HeatingPLC_vAI_Vars".vAI6.iFuncVar);
END_REGION

REGION Network 7
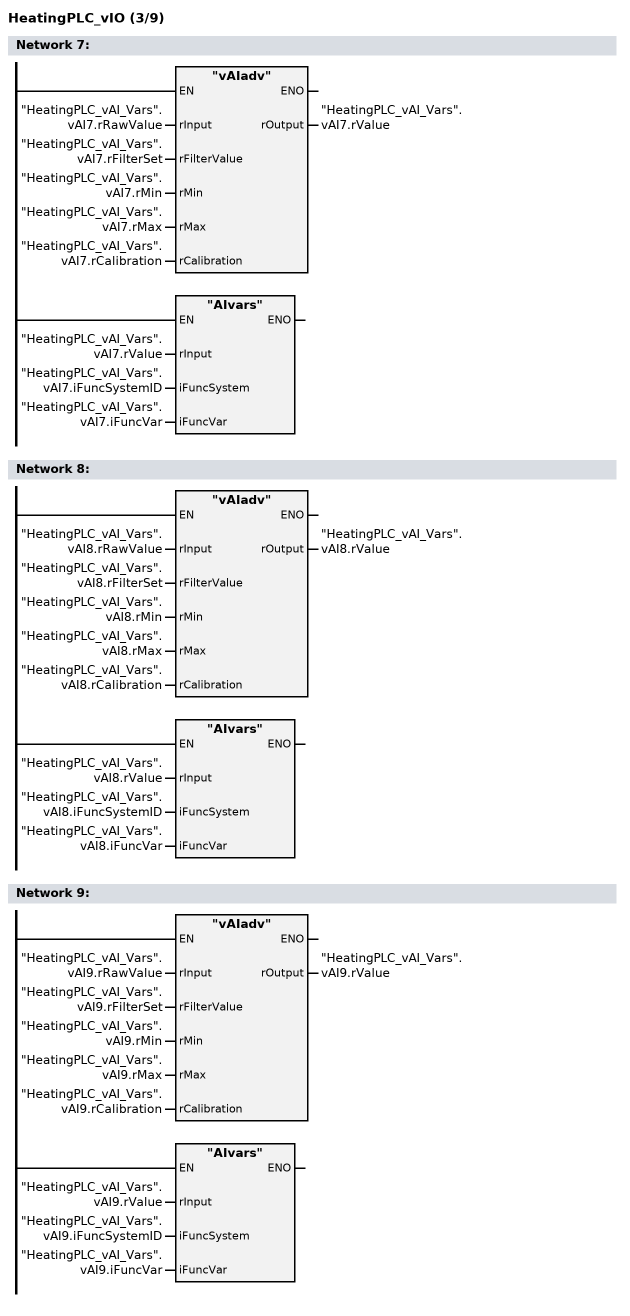
   RUNG wire#powerrail
      "vAIadv"(rInput := "HeatingPLC_vAI_Vars".vAI7.rRawValue, rFilterValue := "HeatingPLC_vAI_Vars".vAI7.rFilterSet, rMin := "HeatingPLC_vAI_Vars".vAI7.rMin, rMax := "HeatingPLC_vAI_Vars".vAI7.rMax, rCalibration := "HeatingPLC_vAI_Vars".vAI7.rCalibration, rOutput => "HeatingPLC_vAI_Vars".vAI7.rValue)
   END_RUNG
   RUNG wire#powerrail
      "AIvars"(rInput := "HeatingPLC_vAI_Vars".vAI7.rValue, iFuncSystem := "HeatingPLC_vAI_Vars".vAI7.iFuncSystemID, iFuncVar := "HeatingPLC_vAI_Vars".vAI7.iFuncVar)
   END_RUNG
   // the same network as SCL:
   "vAIadv"(rInput := "HeatingPLC_vAI_Vars".vAI7.rRawValue,
            rFilterValue := "HeatingPLC_vAI_Vars".vAI7.rFilterSet,
            rMin := "HeatingPLC_vAI_Vars".vAI7.rMin,
            rMax := "HeatingPLC_vAI_Vars".vAI7.rMax,
            rCalibration := "HeatingPLC_vAI_Vars".vAI7.rCalibration,
            rOutput => "HeatingPLC_vAI_Vars".vAI7.rValue);
   "AIvars"(rInput := "HeatingPLC_vAI_Vars".vAI7.rValue,
            iFuncSystem := "HeatingPLC_vAI_Vars".vAI7.iFuncSystemID,
            iFuncVar := "HeatingPLC_vAI_Vars".vAI7.iFuncVar);
END_REGION

REGION Network 8
   RUNG wire#powerrail
      "vAIadv"(rInput := "HeatingPLC_vAI_Vars".vAI8.rRawValue, rFilterValue := "HeatingPLC_vAI_Vars".vAI8.rFilterSet, rMin := "HeatingPLC_vAI_Vars".vAI8.rMin, rMax := "HeatingPLC_vAI_Vars".vAI8.rMax, rCalibration := "HeatingPLC_vAI_Vars".vAI8.rCalibration, rOutput => "HeatingPLC_vAI_Vars".vAI8.rValue)
   END_RUNG
   RUNG wire#powerrail
      "AIvars"(rInput := "HeatingPLC_vAI_Vars".vAI8.rValue, iFuncSystem := "HeatingPLC_vAI_Vars".vAI8.iFuncSystemID, iFuncVar := "HeatingPLC_vAI_Vars".vAI8.iFuncVar)
   END_RUNG
   // the same network as SCL:
   "vAIadv"(rInput := "HeatingPLC_vAI_Vars".vAI8.rRawValue,
            rFilterValue := "HeatingPLC_vAI_Vars".vAI8.rFilterSet,
            rMin := "HeatingPLC_vAI_Vars".vAI8.rMin,
            rMax := "HeatingPLC_vAI_Vars".vAI8.rMax,
            rCalibration := "HeatingPLC_vAI_Vars".vAI8.rCalibration,
            rOutput => "HeatingPLC_vAI_Vars".vAI8.rValue);
   "AIvars"(rInput := "HeatingPLC_vAI_Vars".vAI8.rValue,
            iFuncSystem := "HeatingPLC_vAI_Vars".vAI8.iFuncSystemID,
            iFuncVar := "HeatingPLC_vAI_Vars".vAI8.iFuncVar);
END_REGION

REGION Network 9
   RUNG wire#powerrail
      "vAIadv"(rInput := "HeatingPLC_vAI_Vars".vAI9.rRawValue, rFilterValue := "HeatingPLC_vAI_Vars".vAI9.rFilterSet, rMin := "HeatingPLC_vAI_Vars".vAI9.rMin, rMax := "HeatingPLC_vAI_Vars".vAI9.rMax, rCalibration := "HeatingPLC_vAI_Vars".vAI9.rCalibration, rOutput => "HeatingPLC_vAI_Vars".vAI9.rValue)
   END_RUNG
   RUNG wire#powerrail
      "AIvars"(rInput := "HeatingPLC_vAI_Vars".vAI9.rValue, iFuncSystem := "HeatingPLC_vAI_Vars".vAI9.iFuncSystemID, iFuncVar := "HeatingPLC_vAI_Vars".vAI9.iFuncVar)
   END_RUNG
   // the same network as SCL:
   "vAIadv"(rInput := "HeatingPLC_vAI_Vars".vAI9.rRawValue,
            rFilterValue := "HeatingPLC_vAI_Vars".vAI9.rFilterSet,
            rMin := "HeatingPLC_vAI_Vars".vAI9.rMin,
            rMax := "HeatingPLC_vAI_Vars".vAI9.rMax,
            rCalibration := "HeatingPLC_vAI_Vars".vAI9.rCalibration,
            rOutput => "HeatingPLC_vAI_Vars".vAI9.rValue);
   "AIvars"(rInput := "HeatingPLC_vAI_Vars".vAI9.rValue,
            iFuncSystem := "HeatingPLC_vAI_Vars".vAI9.iFuncSystemID,
            iFuncVar := "HeatingPLC_vAI_Vars".vAI9.iFuncVar);
END_REGION

REGION Network 10
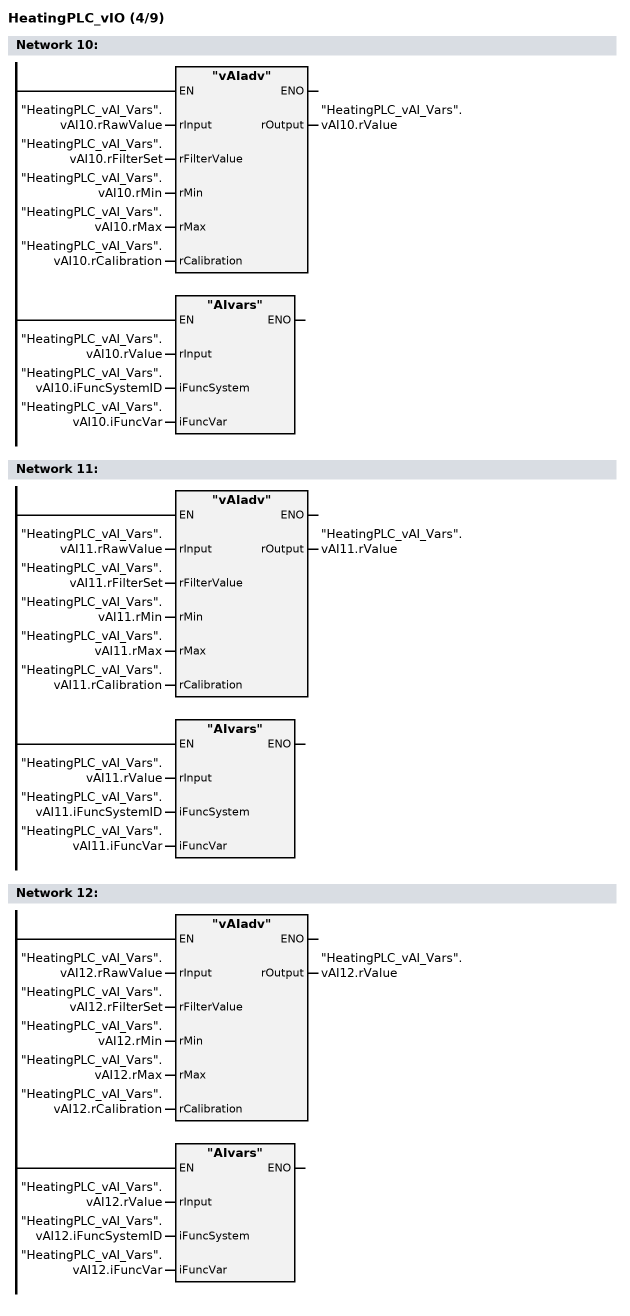
   RUNG wire#powerrail
      "vAIadv"(rInput := "HeatingPLC_vAI_Vars".vAI10.rRawValue, rFilterValue := "HeatingPLC_vAI_Vars".vAI10.rFilterSet, rMin := "HeatingPLC_vAI_Vars".vAI10.rMin, rMax := "HeatingPLC_vAI_Vars".vAI10.rMax, rCalibration := "HeatingPLC_vAI_Vars".vAI10.rCalibration, rOutput => "HeatingPLC_vAI_Vars".vAI10.rValue)
   END_RUNG
   RUNG wire#powerrail
      "AIvars"(rInput := "HeatingPLC_vAI_Vars".vAI10.rValue, iFuncSystem := "HeatingPLC_vAI_Vars".vAI10.iFuncSystemID, iFuncVar := "HeatingPLC_vAI_Vars".vAI10.iFuncVar)
   END_RUNG
   // the same network as SCL:
   "vAIadv"(rInput := "HeatingPLC_vAI_Vars".vAI10.rRawValue,
            rFilterValue := "HeatingPLC_vAI_Vars".vAI10.rFilterSet,
            rMin := "HeatingPLC_vAI_Vars".vAI10.rMin,
            rMax := "HeatingPLC_vAI_Vars".vAI10.rMax,
            rCalibration := "HeatingPLC_vAI_Vars".vAI10.rCalibration,
            rOutput => "HeatingPLC_vAI_Vars".vAI10.rValue);
   "AIvars"(rInput := "HeatingPLC_vAI_Vars".vAI10.rValue,
            iFuncSystem := "HeatingPLC_vAI_Vars".vAI10.iFuncSystemID,
            iFuncVar := "HeatingPLC_vAI_Vars".vAI10.iFuncVar);
END_REGION

REGION Network 11
   RUNG wire#powerrail
      "vAIadv"(rInput := "HeatingPLC_vAI_Vars".vAI11.rRawValue, rFilterValue := "HeatingPLC_vAI_Vars".vAI11.rFilterSet, rMin := "HeatingPLC_vAI_Vars".vAI11.rMin, rMax := "HeatingPLC_vAI_Vars".vAI11.rMax, rCalibration := "HeatingPLC_vAI_Vars".vAI11.rCalibration, rOutput => "HeatingPLC_vAI_Vars".vAI11.rValue)
   END_RUNG
   RUNG wire#powerrail
      "AIvars"(rInput := "HeatingPLC_vAI_Vars".vAI11.rValue, iFuncSystem := "HeatingPLC_vAI_Vars".vAI11.iFuncSystemID, iFuncVar := "HeatingPLC_vAI_Vars".vAI11.iFuncVar)
   END_RUNG
   // the same network as SCL:
   "vAIadv"(rInput := "HeatingPLC_vAI_Vars".vAI11.rRawValue,
            rFilterValue := "HeatingPLC_vAI_Vars".vAI11.rFilterSet,
            rMin := "HeatingPLC_vAI_Vars".vAI11.rMin,
            rMax := "HeatingPLC_vAI_Vars".vAI11.rMax,
            rCalibration := "HeatingPLC_vAI_Vars".vAI11.rCalibration,
            rOutput => "HeatingPLC_vAI_Vars".vAI11.rValue);
   "AIvars"(rInput := "HeatingPLC_vAI_Vars".vAI11.rValue,
            iFuncSystem := "HeatingPLC_vAI_Vars".vAI11.iFuncSystemID,
            iFuncVar := "HeatingPLC_vAI_Vars".vAI11.iFuncVar);
END_REGION

REGION Network 12
   RUNG wire#powerrail
      "vAIadv"(rInput := "HeatingPLC_vAI_Vars".vAI12.rRawValue, rFilterValue := "HeatingPLC_vAI_Vars".vAI12.rFilterSet, rMin := "HeatingPLC_vAI_Vars".vAI12.rMin, rMax := "HeatingPLC_vAI_Vars".vAI12.rMax, rCalibration := "HeatingPLC_vAI_Vars".vAI12.rCalibration, rOutput => "HeatingPLC_vAI_Vars".vAI12.rValue)
   END_RUNG
   RUNG wire#powerrail
      "AIvars"(rInput := "HeatingPLC_vAI_Vars".vAI12.rValue, iFuncSystem := "HeatingPLC_vAI_Vars".vAI12.iFuncSystemID, iFuncVar := "HeatingPLC_vAI_Vars".vAI12.iFuncVar)
   END_RUNG
   // the same network as SCL:
   "vAIadv"(rInput := "HeatingPLC_vAI_Vars".vAI12.rRawValue,
            rFilterValue := "HeatingPLC_vAI_Vars".vAI12.rFilterSet,
            rMin := "HeatingPLC_vAI_Vars".vAI12.rMin,
            rMax := "HeatingPLC_vAI_Vars".vAI12.rMax,
            rCalibration := "HeatingPLC_vAI_Vars".vAI12.rCalibration,
            rOutput => "HeatingPLC_vAI_Vars".vAI12.rValue);
   "AIvars"(rInput := "HeatingPLC_vAI_Vars".vAI12.rValue,
            iFuncSystem := "HeatingPLC_vAI_Vars".vAI12.iFuncSystemID,
            iFuncVar := "HeatingPLC_vAI_Vars".vAI12.iFuncVar);
END_REGION

REGION Network 13
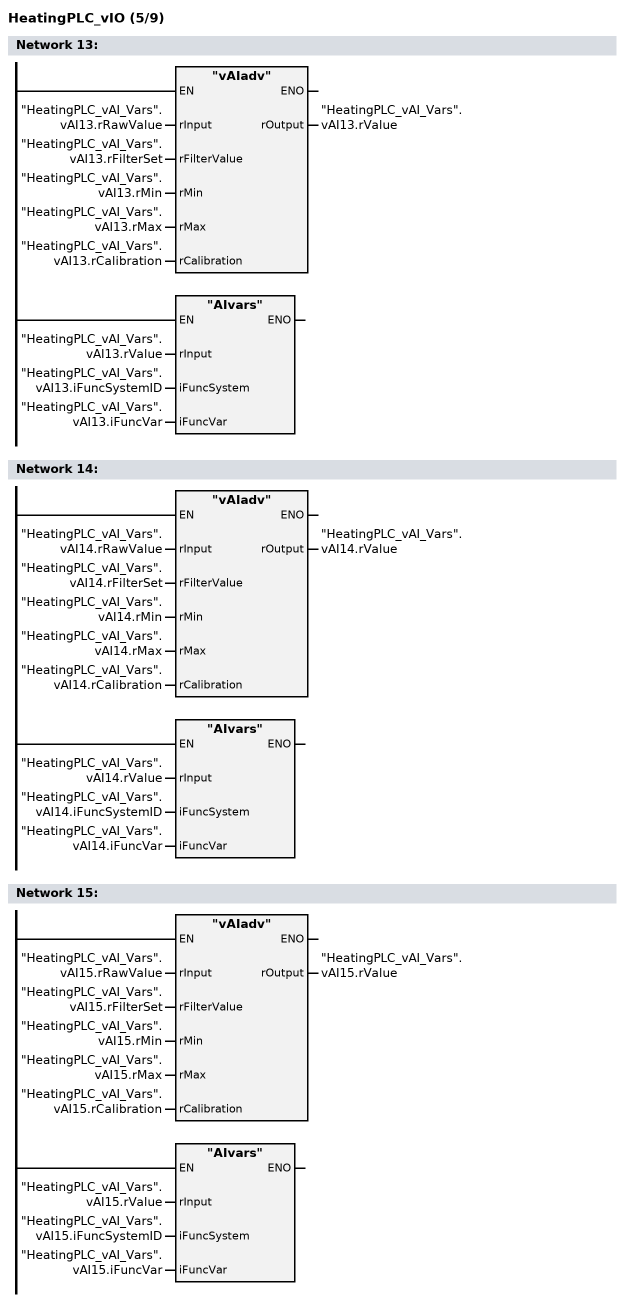
   RUNG wire#powerrail
      "vAIadv"(rInput := "HeatingPLC_vAI_Vars".vAI13.rRawValue, rFilterValue := "HeatingPLC_vAI_Vars".vAI13.rFilterSet, rMin := "HeatingPLC_vAI_Vars".vAI13.rMin, rMax := "HeatingPLC_vAI_Vars".vAI13.rMax, rCalibration := "HeatingPLC_vAI_Vars".vAI13.rCalibration, rOutput => "HeatingPLC_vAI_Vars".vAI13.rValue)
   END_RUNG
   RUNG wire#powerrail
      "AIvars"(rInput := "HeatingPLC_vAI_Vars".vAI13.rValue, iFuncSystem := "HeatingPLC_vAI_Vars".vAI13.iFuncSystemID, iFuncVar := "HeatingPLC_vAI_Vars".vAI13.iFuncVar)
   END_RUNG
   // the same network as SCL:
   "vAIadv"(rInput := "HeatingPLC_vAI_Vars".vAI13.rRawValue,
            rFilterValue := "HeatingPLC_vAI_Vars".vAI13.rFilterSet,
            rMin := "HeatingPLC_vAI_Vars".vAI13.rMin,
            rMax := "HeatingPLC_vAI_Vars".vAI13.rMax,
            rCalibration := "HeatingPLC_vAI_Vars".vAI13.rCalibration,
            rOutput => "HeatingPLC_vAI_Vars".vAI13.rValue);
   "AIvars"(rInput := "HeatingPLC_vAI_Vars".vAI13.rValue,
            iFuncSystem := "HeatingPLC_vAI_Vars".vAI13.iFuncSystemID,
            iFuncVar := "HeatingPLC_vAI_Vars".vAI13.iFuncVar);
END_REGION

REGION Network 14
   RUNG wire#powerrail
      "vAIadv"(rInput := "HeatingPLC_vAI_Vars".vAI14.rRawValue, rFilterValue := "HeatingPLC_vAI_Vars".vAI14.rFilterSet, rMin := "HeatingPLC_vAI_Vars".vAI14.rMin, rMax := "HeatingPLC_vAI_Vars".vAI14.rMax, rCalibration := "HeatingPLC_vAI_Vars".vAI14.rCalibration, rOutput => "HeatingPLC_vAI_Vars".vAI14.rValue)
   END_RUNG
   RUNG wire#powerrail
      "AIvars"(rInput := "HeatingPLC_vAI_Vars".vAI14.rValue, iFuncSystem := "HeatingPLC_vAI_Vars".vAI14.iFuncSystemID, iFuncVar := "HeatingPLC_vAI_Vars".vAI14.iFuncVar)
   END_RUNG
   // the same network as SCL:
   "vAIadv"(rInput := "HeatingPLC_vAI_Vars".vAI14.rRawValue,
            rFilterValue := "HeatingPLC_vAI_Vars".vAI14.rFilterSet,
            rMin := "HeatingPLC_vAI_Vars".vAI14.rMin,
            rMax := "HeatingPLC_vAI_Vars".vAI14.rMax,
            rCalibration := "HeatingPLC_vAI_Vars".vAI14.rCalibration,
            rOutput => "HeatingPLC_vAI_Vars".vAI14.rValue);
   "AIvars"(rInput := "HeatingPLC_vAI_Vars".vAI14.rValue,
            iFuncSystem := "HeatingPLC_vAI_Vars".vAI14.iFuncSystemID,
            iFuncVar := "HeatingPLC_vAI_Vars".vAI14.iFuncVar);
END_REGION

REGION Network 15
   RUNG wire#powerrail
      "vAIadv"(rInput := "HeatingPLC_vAI_Vars".vAI15.rRawValue, rFilterValue := "HeatingPLC_vAI_Vars".vAI15.rFilterSet, rMin := "HeatingPLC_vAI_Vars".vAI15.rMin, rMax := "HeatingPLC_vAI_Vars".vAI15.rMax, rCalibration := "HeatingPLC_vAI_Vars".vAI15.rCalibration, rOutput => "HeatingPLC_vAI_Vars".vAI15.rValue)
   END_RUNG
   RUNG wire#powerrail
      "AIvars"(rInput := "HeatingPLC_vAI_Vars".vAI15.rValue, iFuncSystem := "HeatingPLC_vAI_Vars".vAI15.iFuncSystemID, iFuncVar := "HeatingPLC_vAI_Vars".vAI15.iFuncVar)
   END_RUNG
   // the same network as SCL:
   "vAIadv"(rInput := "HeatingPLC_vAI_Vars".vAI15.rRawValue,
            rFilterValue := "HeatingPLC_vAI_Vars".vAI15.rFilterSet,
            rMin := "HeatingPLC_vAI_Vars".vAI15.rMin,
            rMax := "HeatingPLC_vAI_Vars".vAI15.rMax,
            rCalibration := "HeatingPLC_vAI_Vars".vAI15.rCalibration,
            rOutput => "HeatingPLC_vAI_Vars".vAI15.rValue);
   "AIvars"(rInput := "HeatingPLC_vAI_Vars".vAI15.rValue,
            iFuncSystem := "HeatingPLC_vAI_Vars".vAI15.iFuncSystemID,
            iFuncVar := "HeatingPLC_vAI_Vars".vAI15.iFuncVar);
END_REGION

REGION Network 16
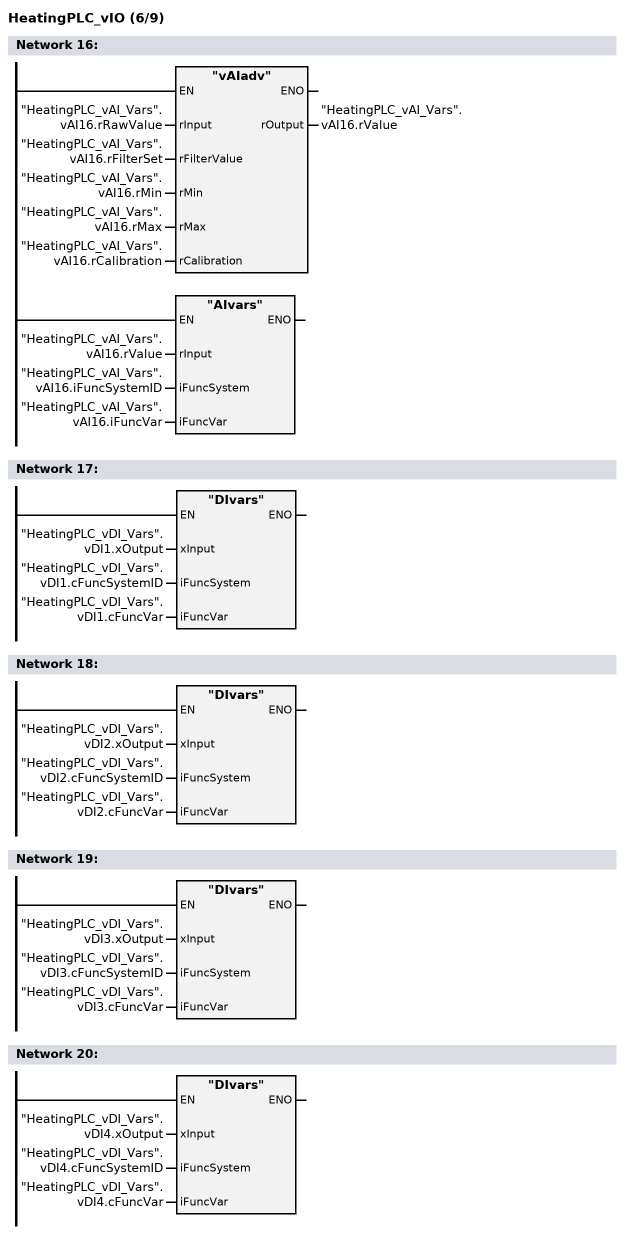
   RUNG wire#powerrail
      "vAIadv"(rInput := "HeatingPLC_vAI_Vars".vAI16.rRawValue, rFilterValue := "HeatingPLC_vAI_Vars".vAI16.rFilterSet, rMin := "HeatingPLC_vAI_Vars".vAI16.rMin, rMax := "HeatingPLC_vAI_Vars".vAI16.rMax, rCalibration := "HeatingPLC_vAI_Vars".vAI16.rCalibration, rOutput => "HeatingPLC_vAI_Vars".vAI16.rValue)
   END_RUNG
   RUNG wire#powerrail
      "AIvars"(rInput := "HeatingPLC_vAI_Vars".vAI16.rValue, iFuncSystem := "HeatingPLC_vAI_Vars".vAI16.iFuncSystemID, iFuncVar := "HeatingPLC_vAI_Vars".vAI16.iFuncVar)
   END_RUNG
   // the same network as SCL:
   "vAIadv"(rInput := "HeatingPLC_vAI_Vars".vAI16.rRawValue,
            rFilterValue := "HeatingPLC_vAI_Vars".vAI16.rFilterSet,
            rMin := "HeatingPLC_vAI_Vars".vAI16.rMin,
            rMax := "HeatingPLC_vAI_Vars".vAI16.rMax,
            rCalibration := "HeatingPLC_vAI_Vars".vAI16.rCalibration,
            rOutput => "HeatingPLC_vAI_Vars".vAI16.rValue);
   "AIvars"(rInput := "HeatingPLC_vAI_Vars".vAI16.rValue,
            iFuncSystem := "HeatingPLC_vAI_Vars".vAI16.iFuncSystemID,
            iFuncVar := "HeatingPLC_vAI_Vars".vAI16.iFuncVar);
END_REGION

REGION Network 17
   RUNG wire#powerrail
      "DIvars"(xInput := "HeatingPLC_vDI_Vars".vDI1.xOutput, iFuncSystem := "HeatingPLC_vDI_Vars".vDI1.cFuncSystemID, iFuncVar := "HeatingPLC_vDI_Vars".vDI1.cFuncVar)
   END_RUNG
   // the same network as SCL:
   "DIvars"(xInput := "HeatingPLC_vDI_Vars".vDI1.xOutput,
            iFuncSystem := "HeatingPLC_vDI_Vars".vDI1.cFuncSystemID,
            iFuncVar := "HeatingPLC_vDI_Vars".vDI1.cFuncVar);
END_REGION

REGION Network 18
   RUNG wire#powerrail
      "DIvars"(xInput := "HeatingPLC_vDI_Vars".vDI2.xOutput, iFuncSystem := "HeatingPLC_vDI_Vars".vDI2.cFuncSystemID, iFuncVar := "HeatingPLC_vDI_Vars".vDI2.cFuncVar)
   END_RUNG
   // the same network as SCL:
   "DIvars"(xInput := "HeatingPLC_vDI_Vars".vDI2.xOutput,
            iFuncSystem := "HeatingPLC_vDI_Vars".vDI2.cFuncSystemID,
            iFuncVar := "HeatingPLC_vDI_Vars".vDI2.cFuncVar);
END_REGION

REGION Network 19
   RUNG wire#powerrail
      "DIvars"(xInput := "HeatingPLC_vDI_Vars".vDI3.xOutput, iFuncSystem := "HeatingPLC_vDI_Vars".vDI3.cFuncSystemID, iFuncVar := "HeatingPLC_vDI_Vars".vDI3.cFuncVar)
   END_RUNG
   // the same network as SCL:
   "DIvars"(xInput := "HeatingPLC_vDI_Vars".vDI3.xOutput,
            iFuncSystem := "HeatingPLC_vDI_Vars".vDI3.cFuncSystemID,
            iFuncVar := "HeatingPLC_vDI_Vars".vDI3.cFuncVar);
END_REGION

REGION Network 20
   RUNG wire#powerrail
      "DIvars"(xInput := "HeatingPLC_vDI_Vars".vDI4.xOutput, iFuncSystem := "HeatingPLC_vDI_Vars".vDI4.cFuncSystemID, iFuncVar := "HeatingPLC_vDI_Vars".vDI4.cFuncVar)
   END_RUNG
   // the same network as SCL:
   "DIvars"(xInput := "HeatingPLC_vDI_Vars".vDI4.xOutput,
            iFuncSystem := "HeatingPLC_vDI_Vars".vDI4.cFuncSystemID,
            iFuncVar := "HeatingPLC_vDI_Vars".vDI4.cFuncVar);
END_REGION

REGION Network 21
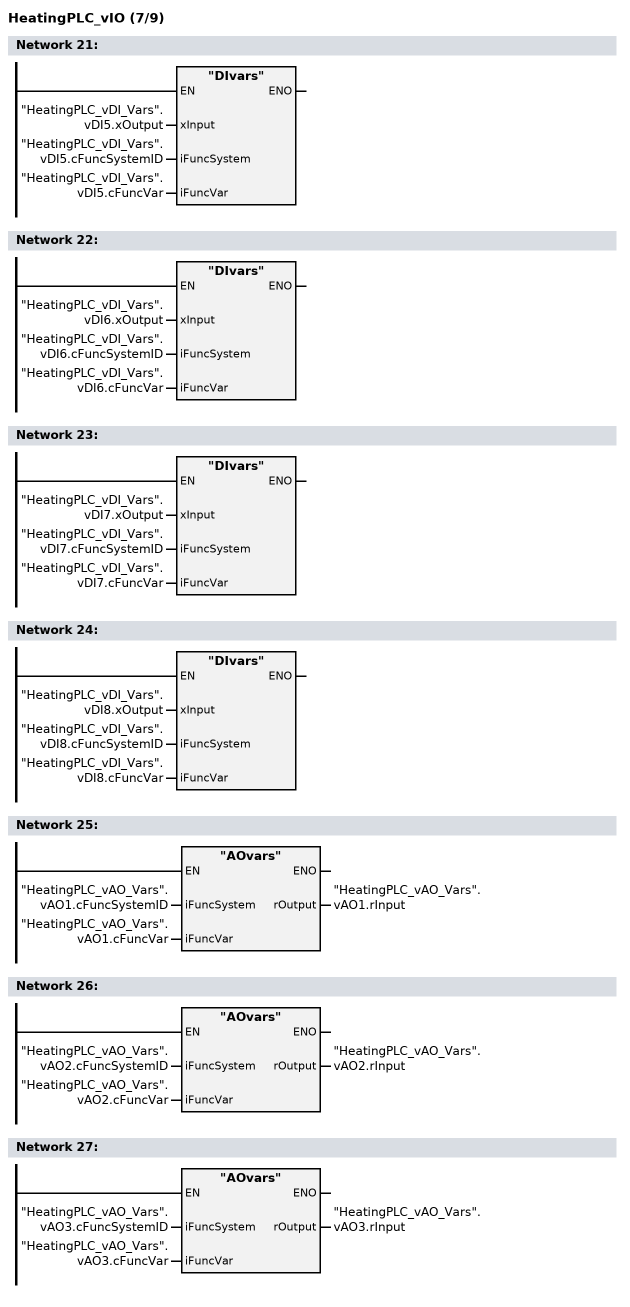
   RUNG wire#powerrail
      "DIvars"(xInput := "HeatingPLC_vDI_Vars".vDI5.xOutput, iFuncSystem := "HeatingPLC_vDI_Vars".vDI5.cFuncSystemID, iFuncVar := "HeatingPLC_vDI_Vars".vDI5.cFuncVar)
   END_RUNG
   // the same network as SCL:
   "DIvars"(xInput := "HeatingPLC_vDI_Vars".vDI5.xOutput,
            iFuncSystem := "HeatingPLC_vDI_Vars".vDI5.cFuncSystemID,
            iFuncVar := "HeatingPLC_vDI_Vars".vDI5.cFuncVar);
END_REGION

REGION Network 22
   RUNG wire#powerrail
      "DIvars"(xInput := "HeatingPLC_vDI_Vars".vDI6.xOutput, iFuncSystem := "HeatingPLC_vDI_Vars".vDI6.cFuncSystemID, iFuncVar := "HeatingPLC_vDI_Vars".vDI6.cFuncVar)
   END_RUNG
   // the same network as SCL:
   "DIvars"(xInput := "HeatingPLC_vDI_Vars".vDI6.xOutput,
            iFuncSystem := "HeatingPLC_vDI_Vars".vDI6.cFuncSystemID,
            iFuncVar := "HeatingPLC_vDI_Vars".vDI6.cFuncVar);
END_REGION

REGION Network 23
   RUNG wire#powerrail
      "DIvars"(xInput := "HeatingPLC_vDI_Vars".vDI7.xOutput, iFuncSystem := "HeatingPLC_vDI_Vars".vDI7.cFuncSystemID, iFuncVar := "HeatingPLC_vDI_Vars".vDI7.cFuncVar)
   END_RUNG
   // the same network as SCL:
   "DIvars"(xInput := "HeatingPLC_vDI_Vars".vDI7.xOutput,
            iFuncSystem := "HeatingPLC_vDI_Vars".vDI7.cFuncSystemID,
            iFuncVar := "HeatingPLC_vDI_Vars".vDI7.cFuncVar);
END_REGION

REGION Network 24
   RUNG wire#powerrail
      "DIvars"(xInput := "HeatingPLC_vDI_Vars".vDI8.xOutput, iFuncSystem := "HeatingPLC_vDI_Vars".vDI8.cFuncSystemID, iFuncVar := "HeatingPLC_vDI_Vars".vDI8.cFuncVar)
   END_RUNG
   // the same network as SCL:
   "DIvars"(xInput := "HeatingPLC_vDI_Vars".vDI8.xOutput,
            iFuncSystem := "HeatingPLC_vDI_Vars".vDI8.cFuncSystemID,
            iFuncVar := "HeatingPLC_vDI_Vars".vDI8.cFuncVar);
END_REGION

REGION Network 25
   RUNG wire#powerrail
      "AOvars"(iFuncSystem := "HeatingPLC_vAO_Vars".vAO1.cFuncSystemID, iFuncVar := "HeatingPLC_vAO_Vars".vAO1.cFuncVar, rOutput => "HeatingPLC_vAO_Vars".vAO1.rInput)
   END_RUNG
   // the same network as SCL:
   "AOvars"(iFuncSystem := "HeatingPLC_vAO_Vars".vAO1.cFuncSystemID,
            iFuncVar := "HeatingPLC_vAO_Vars".vAO1.cFuncVar,
            rOutput => "HeatingPLC_vAO_Vars".vAO1.rInput);
END_REGION

REGION Network 26
   RUNG wire#powerrail
      "AOvars"(iFuncSystem := "HeatingPLC_vAO_Vars".vAO2.cFuncSystemID, iFuncVar := "HeatingPLC_vAO_Vars".vAO2.cFuncVar, rOutput => "HeatingPLC_vAO_Vars".vAO2.rInput)
   END_RUNG
   // the same network as SCL:
   "AOvars"(iFuncSystem := "HeatingPLC_vAO_Vars".vAO2.cFuncSystemID,
            iFuncVar := "HeatingPLC_vAO_Vars".vAO2.cFuncVar,
            rOutput => "HeatingPLC_vAO_Vars".vAO2.rInput);
END_REGION

REGION Network 27
   RUNG wire#powerrail
      "AOvars"(iFuncSystem := "HeatingPLC_vAO_Vars".vAO3.cFuncSystemID, iFuncVar := "HeatingPLC_vAO_Vars".vAO3.cFuncVar, rOutput => "HeatingPLC_vAO_Vars".vAO3.rInput)
   END_RUNG
   // the same network as SCL:
   "AOvars"(iFuncSystem := "HeatingPLC_vAO_Vars".vAO3.cFuncSystemID,
            iFuncVar := "HeatingPLC_vAO_Vars".vAO3.cFuncVar,
            rOutput => "HeatingPLC_vAO_Vars".vAO3.rInput);
END_REGION

REGION Network 28
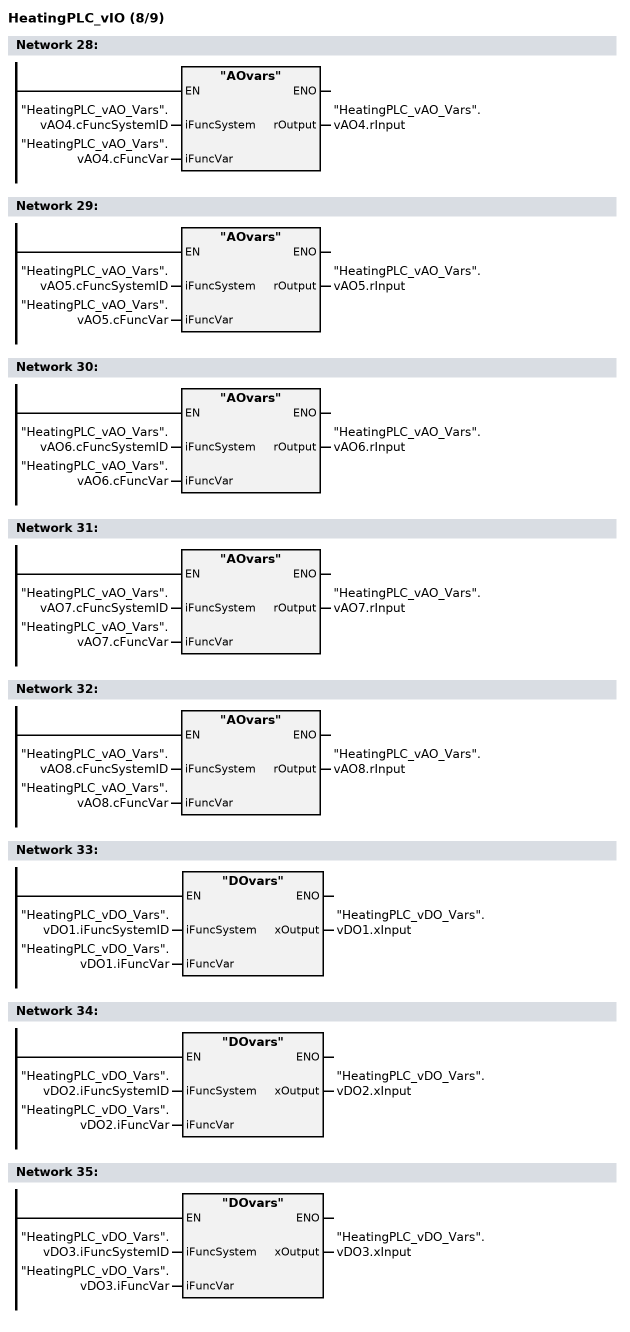
   RUNG wire#powerrail
      "AOvars"(iFuncSystem := "HeatingPLC_vAO_Vars".vAO4.cFuncSystemID, iFuncVar := "HeatingPLC_vAO_Vars".vAO4.cFuncVar, rOutput => "HeatingPLC_vAO_Vars".vAO4.rInput)
   END_RUNG
   // the same network as SCL:
   "AOvars"(iFuncSystem := "HeatingPLC_vAO_Vars".vAO4.cFuncSystemID,
            iFuncVar := "HeatingPLC_vAO_Vars".vAO4.cFuncVar,
            rOutput => "HeatingPLC_vAO_Vars".vAO4.rInput);
END_REGION

REGION Network 29
   RUNG wire#powerrail
      "AOvars"(iFuncSystem := "HeatingPLC_vAO_Vars".vAO5.cFuncSystemID, iFuncVar := "HeatingPLC_vAO_Vars".vAO5.cFuncVar, rOutput => "HeatingPLC_vAO_Vars".vAO5.rInput)
   END_RUNG
   // the same network as SCL:
   "AOvars"(iFuncSystem := "HeatingPLC_vAO_Vars".vAO5.cFuncSystemID,
            iFuncVar := "HeatingPLC_vAO_Vars".vAO5.cFuncVar,
            rOutput => "HeatingPLC_vAO_Vars".vAO5.rInput);
END_REGION

REGION Network 30
   RUNG wire#powerrail
      "AOvars"(iFuncSystem := "HeatingPLC_vAO_Vars".vAO6.cFuncSystemID, iFuncVar := "HeatingPLC_vAO_Vars".vAO6.cFuncVar, rOutput => "HeatingPLC_vAO_Vars".vAO6.rInput)
   END_RUNG
   // the same network as SCL:
   "AOvars"(iFuncSystem := "HeatingPLC_vAO_Vars".vAO6.cFuncSystemID,
            iFuncVar := "HeatingPLC_vAO_Vars".vAO6.cFuncVar,
            rOutput => "HeatingPLC_vAO_Vars".vAO6.rInput);
END_REGION

REGION Network 31
   RUNG wire#powerrail
      "AOvars"(iFuncSystem := "HeatingPLC_vAO_Vars".vAO7.cFuncSystemID, iFuncVar := "HeatingPLC_vAO_Vars".vAO7.cFuncVar, rOutput => "HeatingPLC_vAO_Vars".vAO7.rInput)
   END_RUNG
   // the same network as SCL:
   "AOvars"(iFuncSystem := "HeatingPLC_vAO_Vars".vAO7.cFuncSystemID,
            iFuncVar := "HeatingPLC_vAO_Vars".vAO7.cFuncVar,
            rOutput => "HeatingPLC_vAO_Vars".vAO7.rInput);
END_REGION

REGION Network 32
   RUNG wire#powerrail
      "AOvars"(iFuncSystem := "HeatingPLC_vAO_Vars".vAO8.cFuncSystemID, iFuncVar := "HeatingPLC_vAO_Vars".vAO8.cFuncVar, rOutput => "HeatingPLC_vAO_Vars".vAO8.rInput)
   END_RUNG
   // the same network as SCL:
   "AOvars"(iFuncSystem := "HeatingPLC_vAO_Vars".vAO8.cFuncSystemID,
            iFuncVar := "HeatingPLC_vAO_Vars".vAO8.cFuncVar,
            rOutput => "HeatingPLC_vAO_Vars".vAO8.rInput);
END_REGION

REGION Network 33
   RUNG wire#powerrail
      "DOvars"(iFuncSystem := "HeatingPLC_vDO_Vars".vDO1.iFuncSystemID, iFuncVar := "HeatingPLC_vDO_Vars".vDO1.iFuncVar, xOutput => "HeatingPLC_vDO_Vars".vDO1.xInput)
   END_RUNG
   // the same network as SCL:
   "DOvars"(iFuncSystem := "HeatingPLC_vDO_Vars".vDO1.iFuncSystemID,
            iFuncVar := "HeatingPLC_vDO_Vars".vDO1.iFuncVar,
            xOutput => "HeatingPLC_vDO_Vars".vDO1.xInput);
END_REGION

REGION Network 34
   RUNG wire#powerrail
      "DOvars"(iFuncSystem := "HeatingPLC_vDO_Vars".vDO2.iFuncSystemID, iFuncVar := "HeatingPLC_vDO_Vars".vDO2.iFuncVar, xOutput => "HeatingPLC_vDO_Vars".vDO2.xInput)
   END_RUNG
   // the same network as SCL:
   "DOvars"(iFuncSystem := "HeatingPLC_vDO_Vars".vDO2.iFuncSystemID,
            iFuncVar := "HeatingPLC_vDO_Vars".vDO2.iFuncVar,
            xOutput => "HeatingPLC_vDO_Vars".vDO2.xInput);
END_REGION

REGION Network 35
   RUNG wire#powerrail
      "DOvars"(iFuncSystem := "HeatingPLC_vDO_Vars".vDO3.iFuncSystemID, iFuncVar := "HeatingPLC_vDO_Vars".vDO3.iFuncVar, xOutput => "HeatingPLC_vDO_Vars".vDO3.xInput)
   END_RUNG
   // the same network as SCL:
   "DOvars"(iFuncSystem := "HeatingPLC_vDO_Vars".vDO3.iFuncSystemID,
            iFuncVar := "HeatingPLC_vDO_Vars".vDO3.iFuncVar,
            xOutput => "HeatingPLC_vDO_Vars".vDO3.xInput);
END_REGION

REGION Network 36
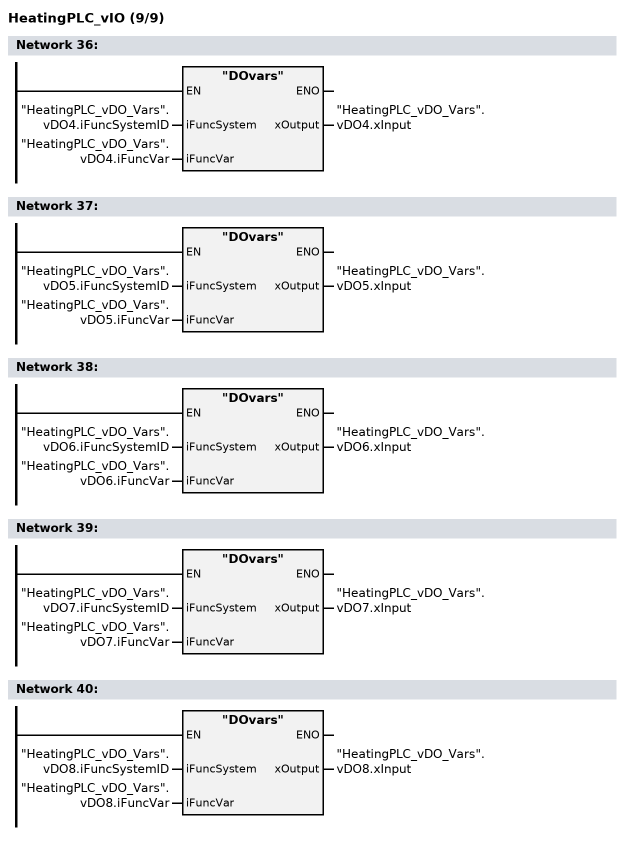
   RUNG wire#powerrail
      "DOvars"(iFuncSystem := "HeatingPLC_vDO_Vars".vDO4.iFuncSystemID, iFuncVar := "HeatingPLC_vDO_Vars".vDO4.iFuncVar, xOutput => "HeatingPLC_vDO_Vars".vDO4.xInput)
   END_RUNG
   // the same network as SCL:
   "DOvars"(iFuncSystem := "HeatingPLC_vDO_Vars".vDO4.iFuncSystemID,
            iFuncVar := "HeatingPLC_vDO_Vars".vDO4.iFuncVar,
            xOutput => "HeatingPLC_vDO_Vars".vDO4.xInput);
END_REGION

REGION Network 37
   RUNG wire#powerrail
      "DOvars"(iFuncSystem := "HeatingPLC_vDO_Vars".vDO5.iFuncSystemID, iFuncVar := "HeatingPLC_vDO_Vars".vDO5.iFuncVar, xOutput => "HeatingPLC_vDO_Vars".vDO5.xInput)
   END_RUNG
   // the same network as SCL:
   "DOvars"(iFuncSystem := "HeatingPLC_vDO_Vars".vDO5.iFuncSystemID,
            iFuncVar := "HeatingPLC_vDO_Vars".vDO5.iFuncVar,
            xOutput => "HeatingPLC_vDO_Vars".vDO5.xInput);
END_REGION

REGION Network 38
   RUNG wire#powerrail
      "DOvars"(iFuncSystem := "HeatingPLC_vDO_Vars".vDO6.iFuncSystemID, iFuncVar := "HeatingPLC_vDO_Vars".vDO6.iFuncVar, xOutput => "HeatingPLC_vDO_Vars".vDO6.xInput)
   END_RUNG
   // the same network as SCL:
   "DOvars"(iFuncSystem := "HeatingPLC_vDO_Vars".vDO6.iFuncSystemID,
            iFuncVar := "HeatingPLC_vDO_Vars".vDO6.iFuncVar,
            xOutput => "HeatingPLC_vDO_Vars".vDO6.xInput);
END_REGION

REGION Network 39
   RUNG wire#powerrail
      "DOvars"(iFuncSystem := "HeatingPLC_vDO_Vars".vDO7.iFuncSystemID, iFuncVar := "HeatingPLC_vDO_Vars".vDO7.iFuncVar, xOutput => "HeatingPLC_vDO_Vars".vDO7.xInput)
   END_RUNG
   // the same network as SCL:
   "DOvars"(iFuncSystem := "HeatingPLC_vDO_Vars".vDO7.iFuncSystemID,
            iFuncVar := "HeatingPLC_vDO_Vars".vDO7.iFuncVar,
            xOutput => "HeatingPLC_vDO_Vars".vDO7.xInput);
END_REGION

REGION Network 40
   RUNG wire#powerrail
      "DOvars"(iFuncSystem := "HeatingPLC_vDO_Vars".vDO8.iFuncSystemID, iFuncVar := "HeatingPLC_vDO_Vars".vDO8.iFuncVar, xOutput => "HeatingPLC_vDO_Vars".vDO8.xInput)
   END_RUNG
   // the same network as SCL:
   "DOvars"(iFuncSystem := "HeatingPLC_vDO_Vars".vDO8.iFuncSystemID,
            iFuncVar := "HeatingPLC_vDO_Vars".vDO8.iFuncVar,
            xOutput => "HeatingPLC_vDO_Vars".vDO8.xInput);
END_REGION
END_FUNCTION

FUNCTION "AOvars" : Void   // FC10011, LAD
{ S7_Optimized_Access := 'TRUE' }
VERSION : 0.1
// stored: AutoNumber false, IsIECCheckEnabled false, SetENOAutomatically false, UDAEnableTagReadback false
   VAR_INPUT
      iFuncSystem : Byte;
      iFuncVar : Byte;
   END_VAR
   VAR_OUTPUT
      rOutput : Real;
   END_VAR
BEGIN

REGION Network 1 (SCL)
   CASE #iFuncSystem OF
       0:  // Statement section case 2 to 4
           ;
       1..4:  // Statement section case 1
           CASE #iFuncVar OF
               0:  // 
                   ;
               1:  // 
                   #rOutput := "AHUAO".AO.rSAFAnalog[#iFuncSystem];
               2:  // 
                   #rOutput := "AHUAO".AO.rHeater[#iFuncSystem];
               3:  // 
                   #rOutput := "AHUAO".AO.rMixingAirDumper[#iFuncSystem];
               4:  // 
                   #rOutput := "AHUAO".AO.rExtractAirDumper[#iFuncSystem];
               5:  // 
                   #rOutput := "AHUAO".AO.rCooler[#iFuncSystem];
               6:  // 
                   #rOutput := "AHUAO".AO.rWHU[#iFuncSystem];
           END_CASE;
       5..9:
           ;
       10: // HS+HC    
           CASE #iFuncVar OF
               0:  // 
                   ;
               1:  //         
                   #rOutput := "HCsAO".AO.rHC3vwCtrl[1];
               2:  //         
                   #rOutput := "HCsAO".AO.rHC3vwCtrl[2];
           END_CASE;
       11..20:
           ;
       21: //Proxy Channels    
           CASE #iFuncVar OF
               0:  //
                   ;
               1..8:  //
                   #rOutput := "AHUProxyCH".Vars.rCHProxySignal[#iFuncVar];
               ELSE
                   ;
           END_CASE;
       ELSE  // Statement section ELSE
           ;
   END_CASE;
END_REGION
END_FUNCTION

FUNCTION "DOvars" : Void   // FC10010, LAD
{ S7_Optimized_Access := 'TRUE' }
VERSION : 0.1
// stored: AutoNumber false, IsIECCheckEnabled false, SetENOAutomatically false, UDAEnableTagReadback false
   VAR_INPUT
      iFuncSystem : Byte;
      iFuncVar : Byte;
   END_VAR
   VAR_OUTPUT
      xOutput : Bool;
   END_VAR
BEGIN

REGION Network 1 (SCL)
   CASE #iFuncSystem OF
       0:  // Statement section case 2 to 4
           ;
       1..4:  // Statement section case 1
           CASE #iFuncVar OF
               0:  // 
                   ;
               1:  // 
                   #xOutput := "AHUDO".Requests.xHeaterPumpCmd[#iFuncSystem];
               2:  // 
                   #xOutput := "AHUDO".Requests.xSAFAnalogEnable[#iFuncSystem];
               3:  // 
                   #xOutput := "AHUDO".Requests.xSAFSp1Cmd[#iFuncSystem];
               4:  // 
                   #xOutput := "AHUDO".Requests.xSAFSp2Cmd[#iFuncSystem];
               5:  // 
                   #xOutput := "AHUDO".Requests.xCoolerSt1Cmd[#iFuncSystem];
               6:  // 
                   #xOutput := "AHUDO".Requests.xCoolerSt2Cmd[#iFuncSystem];
               7:  // 
                   #xOutput := "AHUDO".Requests.xCoolerSt3Cmd[#iFuncSystem];
               8:  // 
                   #xOutput := "AHUDO".Requests.xCoolerSt4Cmd[#iFuncSystem];
           END_CASE;
       5:
           ;
       6:
           ;
       7:  // AirCond    
           CASE #iFuncVar OF
               0:  // 
                   ;
               1:  // 
                   #xOutput := "ACDO".Requests.xACCentralEnable;
           END_CASE;
       8:  // AirHeaters
           CASE #iFuncVar OF
               0:  // 
                   ;
               1:  // 
                   #xOutput := "AHDO".Requests.xAHCentralEnable;
           END_CASE;
       9:
           ;
       10:
           CASE #iFuncVar OF
               0:  // 
                   ;
               1:  // 
                   #xOutput := "HCsDO".Requests.xHC3wvIncrease[1];
               2:  // 
                   #xOutput := "HCsDO".Requests.xHC3wvDecrease[1];
               3:  // 
                   #xOutput := "HCsDO".Requests.xHC3wvIncrease[2];
               4:  // 
                   #xOutput := "HCsDO".Requests.xHC3wvDecrease[2];
               5:  //
                   #xOutput := "HCsDO".Requests.xHCPump1Cmd[1];
               6:  //
                   #xOutput := "HCsDO".Requests.xHCPump2Cmd[1];
               7:  //
                   #xOutput := "HCsDO".Requests.xHCPump1Cmd[2];
               8:  //
                   #xOutput := "HCsDO".Requests.xHCPump2Cmd[2];
               9:  //    
                   ;
               10:
                   #xOutput := "HSsDO".Requests.xBoilerEnable[1];
               11:
                   #xOutput := "HSsDO".Requests.xBoilerSt1Enable[1];
               12:
                   #xOutput := "HSsDO".Requests.xBoilerSt2Enable[1];
               13:
                   #xOutput := "HSsDO".Requests.xBoilerShuntPumpEnable[1];
               14:
                   #xOutput := "HSsDO".Requests.xBoilerShutOffValveCmd[1];
               15:
                   ;
               16:
                   #xOutput := "HSsDO".Requests.xBoilerEnable[2];
               17:
                   #xOutput := "HSsDO".Requests.xBoilerSt1Enable[2];
               18:
                   #xOutput := "HSsDO".Requests.xBoilerSt2Enable[2];
               19:
                   #xOutput := "HSsDO".Requests.xBoilerShuntPumpEnable[2];
               20:
                   #xOutput := "HSsDO".Requests.xBoilerShutOffValveCmd[2];
               ELSE:
                   ;
           END_CASE;
       11..99:
           ;
       100:    //DieselLine
           CASE #iFuncVar OF
               0:  // 
                   ;
               1:  // 
                   #xOutput := "DLsDO".Requests.xDieselLineHeatingCmd[1];
               2:  // 
                   #xOutput := "DLsDO".Requests.xDieselLineHeatingCmd[2];
               3:  // 
                   #xOutput := "DLsDO".Requests.xDieselLinePumpEnable;
               4:  // 
                   #xOutput := "DLsDO".Requests.xDieselLinePumpSelect;
               5:  //
                   #xOutput := "DLsDO".Requests.xDieselLineDayTankValve[1];
               6:  //
                   #xOutput := "DLsDO".Requests.xDieselLineDayTankValve[2];
               ELSE:
                   ;
           END_CASE;
       ELSE  // Statement section ELSE
           ;
   END_CASE;
END_REGION
END_FUNCTION

FUNCTION "SS1_A2_8RTD_IO_Update" : Void   // FC11020, LAD
{ S7_Optimized_Access := 'TRUE' }
VERSION : 0.1
// stored: AutoNumber false, IsIECCheckEnabled false, SetENOAutomatically false, UDAEnableTagReadback false
BEGIN

REGION Network 1
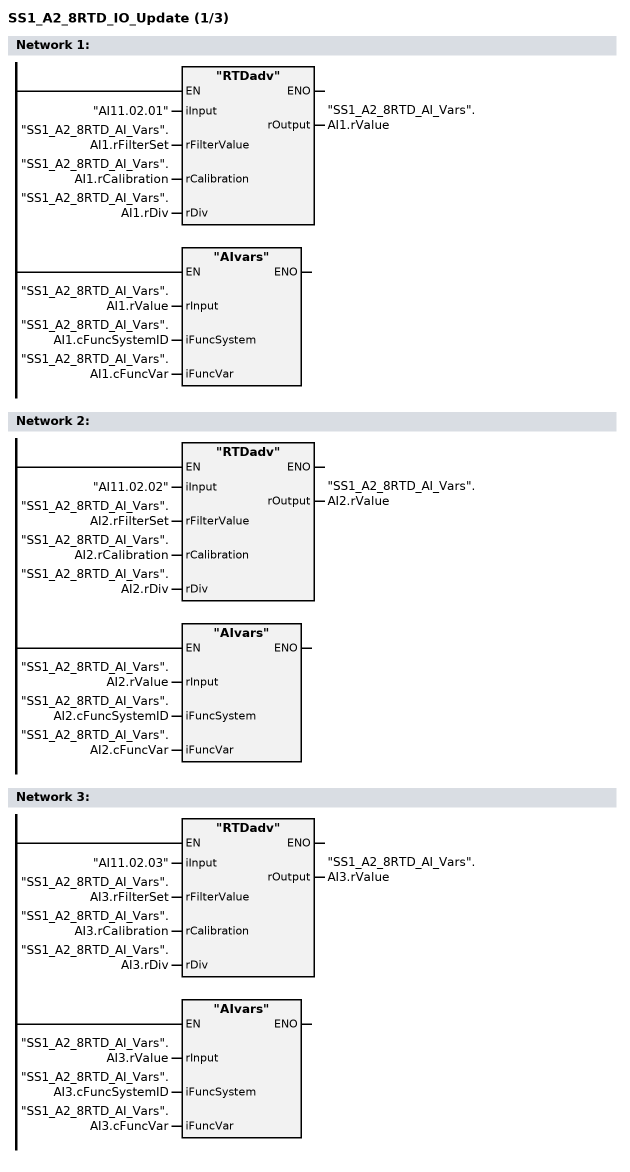
   RUNG wire#powerrail
      "RTDadv"(iInput := "AI11.02.01", rFilterValue := "SS1_A2_8RTD_AI_Vars".AI1.rFilterSet, rCalibration := "SS1_A2_8RTD_AI_Vars".AI1.rCalibration, rDiv := "SS1_A2_8RTD_AI_Vars".AI1.rDiv, rOutput => "SS1_A2_8RTD_AI_Vars".AI1.rValue)
   END_RUNG
   RUNG wire#powerrail
      "AIvars"(rInput := "SS1_A2_8RTD_AI_Vars".AI1.rValue, iFuncSystem := "SS1_A2_8RTD_AI_Vars".AI1.cFuncSystemID, iFuncVar := "SS1_A2_8RTD_AI_Vars".AI1.cFuncVar)
   END_RUNG
   // the same network as SCL:
   "RTDadv"(iInput := "AI11.02.01",
            rFilterValue := "SS1_A2_8RTD_AI_Vars".AI1.rFilterSet,
            rCalibration := "SS1_A2_8RTD_AI_Vars".AI1.rCalibration,
            rDiv := "SS1_A2_8RTD_AI_Vars".AI1.rDiv,
            rOutput => "SS1_A2_8RTD_AI_Vars".AI1.rValue);
   "AIvars"(rInput := "SS1_A2_8RTD_AI_Vars".AI1.rValue,
            iFuncSystem := "SS1_A2_8RTD_AI_Vars".AI1.cFuncSystemID,
            iFuncVar := "SS1_A2_8RTD_AI_Vars".AI1.cFuncVar);
END_REGION

REGION Network 2
   RUNG wire#powerrail
      "RTDadv"(iInput := "AI11.02.02", rFilterValue := "SS1_A2_8RTD_AI_Vars".AI2.rFilterSet, rCalibration := "SS1_A2_8RTD_AI_Vars".AI2.rCalibration, rDiv := "SS1_A2_8RTD_AI_Vars".AI2.rDiv, rOutput => "SS1_A2_8RTD_AI_Vars".AI2.rValue)
   END_RUNG
   RUNG wire#powerrail
      "AIvars"(rInput := "SS1_A2_8RTD_AI_Vars".AI2.rValue, iFuncSystem := "SS1_A2_8RTD_AI_Vars".AI2.cFuncSystemID, iFuncVar := "SS1_A2_8RTD_AI_Vars".AI2.cFuncVar)
   END_RUNG
   // the same network as SCL:
   "RTDadv"(iInput := "AI11.02.02",
            rFilterValue := "SS1_A2_8RTD_AI_Vars".AI2.rFilterSet,
            rCalibration := "SS1_A2_8RTD_AI_Vars".AI2.rCalibration,
            rDiv := "SS1_A2_8RTD_AI_Vars".AI2.rDiv,
            rOutput => "SS1_A2_8RTD_AI_Vars".AI2.rValue);
   "AIvars"(rInput := "SS1_A2_8RTD_AI_Vars".AI2.rValue,
            iFuncSystem := "SS1_A2_8RTD_AI_Vars".AI2.cFuncSystemID,
            iFuncVar := "SS1_A2_8RTD_AI_Vars".AI2.cFuncVar);
END_REGION

REGION Network 3
   RUNG wire#powerrail
      "RTDadv"(iInput := "AI11.02.03", rFilterValue := "SS1_A2_8RTD_AI_Vars".AI3.rFilterSet, rCalibration := "SS1_A2_8RTD_AI_Vars".AI3.rCalibration, rDiv := "SS1_A2_8RTD_AI_Vars".AI3.rDiv, rOutput => "SS1_A2_8RTD_AI_Vars".AI3.rValue)
   END_RUNG
   RUNG wire#powerrail
      "AIvars"(rInput := "SS1_A2_8RTD_AI_Vars".AI3.rValue, iFuncSystem := "SS1_A2_8RTD_AI_Vars".AI3.cFuncSystemID, iFuncVar := "SS1_A2_8RTD_AI_Vars".AI3.cFuncVar)
   END_RUNG
   // the same network as SCL:
   "RTDadv"(iInput := "AI11.02.03",
            rFilterValue := "SS1_A2_8RTD_AI_Vars".AI3.rFilterSet,
            rCalibration := "SS1_A2_8RTD_AI_Vars".AI3.rCalibration,
            rDiv := "SS1_A2_8RTD_AI_Vars".AI3.rDiv,
            rOutput => "SS1_A2_8RTD_AI_Vars".AI3.rValue);
   "AIvars"(rInput := "SS1_A2_8RTD_AI_Vars".AI3.rValue,
            iFuncSystem := "SS1_A2_8RTD_AI_Vars".AI3.cFuncSystemID,
            iFuncVar := "SS1_A2_8RTD_AI_Vars".AI3.cFuncVar);
END_REGION

REGION Network 4
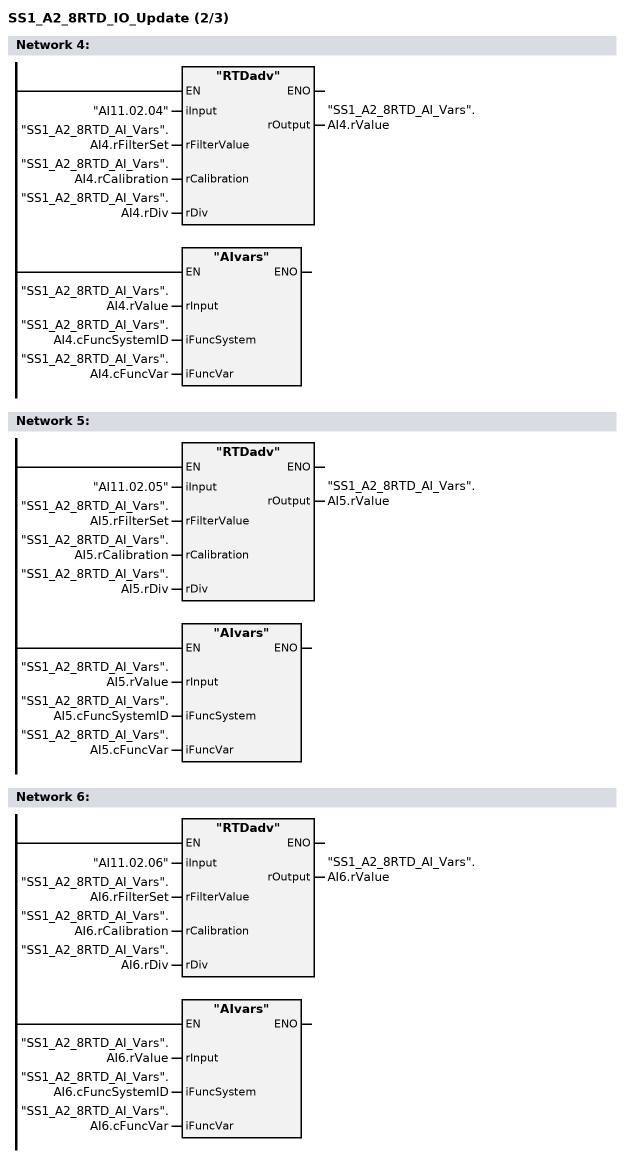
   RUNG wire#powerrail
      "RTDadv"(iInput := "AI11.02.04", rFilterValue := "SS1_A2_8RTD_AI_Vars".AI4.rFilterSet, rCalibration := "SS1_A2_8RTD_AI_Vars".AI4.rCalibration, rDiv := "SS1_A2_8RTD_AI_Vars".AI4.rDiv, rOutput => "SS1_A2_8RTD_AI_Vars".AI4.rValue)
   END_RUNG
   RUNG wire#powerrail
      "AIvars"(rInput := "SS1_A2_8RTD_AI_Vars".AI4.rValue, iFuncSystem := "SS1_A2_8RTD_AI_Vars".AI4.cFuncSystemID, iFuncVar := "SS1_A2_8RTD_AI_Vars".AI4.cFuncVar)
   END_RUNG
   // the same network as SCL:
   "RTDadv"(iInput := "AI11.02.04",
            rFilterValue := "SS1_A2_8RTD_AI_Vars".AI4.rFilterSet,
            rCalibration := "SS1_A2_8RTD_AI_Vars".AI4.rCalibration,
            rDiv := "SS1_A2_8RTD_AI_Vars".AI4.rDiv,
            rOutput => "SS1_A2_8RTD_AI_Vars".AI4.rValue);
   "AIvars"(rInput := "SS1_A2_8RTD_AI_Vars".AI4.rValue,
            iFuncSystem := "SS1_A2_8RTD_AI_Vars".AI4.cFuncSystemID,
            iFuncVar := "SS1_A2_8RTD_AI_Vars".AI4.cFuncVar);
END_REGION

REGION Network 5
   RUNG wire#powerrail
      "RTDadv"(iInput := "AI11.02.05", rFilterValue := "SS1_A2_8RTD_AI_Vars".AI5.rFilterSet, rCalibration := "SS1_A2_8RTD_AI_Vars".AI5.rCalibration, rDiv := "SS1_A2_8RTD_AI_Vars".AI5.rDiv, rOutput => "SS1_A2_8RTD_AI_Vars".AI5.rValue)
   END_RUNG
   RUNG wire#powerrail
      "AIvars"(rInput := "SS1_A2_8RTD_AI_Vars".AI5.rValue, iFuncSystem := "SS1_A2_8RTD_AI_Vars".AI5.cFuncSystemID, iFuncVar := "SS1_A2_8RTD_AI_Vars".AI5.cFuncVar)
   END_RUNG
   // the same network as SCL:
   "RTDadv"(iInput := "AI11.02.05",
            rFilterValue := "SS1_A2_8RTD_AI_Vars".AI5.rFilterSet,
            rCalibration := "SS1_A2_8RTD_AI_Vars".AI5.rCalibration,
            rDiv := "SS1_A2_8RTD_AI_Vars".AI5.rDiv,
            rOutput => "SS1_A2_8RTD_AI_Vars".AI5.rValue);
   "AIvars"(rInput := "SS1_A2_8RTD_AI_Vars".AI5.rValue,
            iFuncSystem := "SS1_A2_8RTD_AI_Vars".AI5.cFuncSystemID,
            iFuncVar := "SS1_A2_8RTD_AI_Vars".AI5.cFuncVar);
END_REGION

REGION Network 6
   RUNG wire#powerrail
      "RTDadv"(iInput := "AI11.02.06", rFilterValue := "SS1_A2_8RTD_AI_Vars".AI6.rFilterSet, rCalibration := "SS1_A2_8RTD_AI_Vars".AI6.rCalibration, rDiv := "SS1_A2_8RTD_AI_Vars".AI6.rDiv, rOutput => "SS1_A2_8RTD_AI_Vars".AI6.rValue)
   END_RUNG
   RUNG wire#powerrail
      "AIvars"(rInput := "SS1_A2_8RTD_AI_Vars".AI6.rValue, iFuncSystem := "SS1_A2_8RTD_AI_Vars".AI6.cFuncSystemID, iFuncVar := "SS1_A2_8RTD_AI_Vars".AI6.cFuncVar)
   END_RUNG
   // the same network as SCL:
   "RTDadv"(iInput := "AI11.02.06",
            rFilterValue := "SS1_A2_8RTD_AI_Vars".AI6.rFilterSet,
            rCalibration := "SS1_A2_8RTD_AI_Vars".AI6.rCalibration,
            rDiv := "SS1_A2_8RTD_AI_Vars".AI6.rDiv,
            rOutput => "SS1_A2_8RTD_AI_Vars".AI6.rValue);
   "AIvars"(rInput := "SS1_A2_8RTD_AI_Vars".AI6.rValue,
            iFuncSystem := "SS1_A2_8RTD_AI_Vars".AI6.cFuncSystemID,
            iFuncVar := "SS1_A2_8RTD_AI_Vars".AI6.cFuncVar);
END_REGION

REGION Network 7
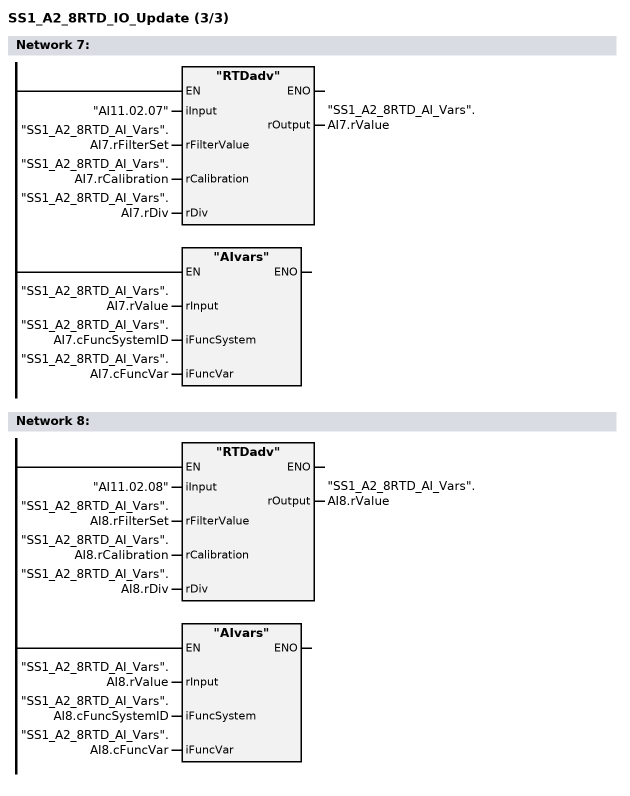
   RUNG wire#powerrail
      "RTDadv"(iInput := "AI11.02.07", rFilterValue := "SS1_A2_8RTD_AI_Vars".AI7.rFilterSet, rCalibration := "SS1_A2_8RTD_AI_Vars".AI7.rCalibration, rDiv := "SS1_A2_8RTD_AI_Vars".AI7.rDiv, rOutput => "SS1_A2_8RTD_AI_Vars".AI7.rValue)
   END_RUNG
   RUNG wire#powerrail
      "AIvars"(rInput := "SS1_A2_8RTD_AI_Vars".AI7.rValue, iFuncSystem := "SS1_A2_8RTD_AI_Vars".AI7.cFuncSystemID, iFuncVar := "SS1_A2_8RTD_AI_Vars".AI7.cFuncVar)
   END_RUNG
   // the same network as SCL:
   "RTDadv"(iInput := "AI11.02.07",
            rFilterValue := "SS1_A2_8RTD_AI_Vars".AI7.rFilterSet,
            rCalibration := "SS1_A2_8RTD_AI_Vars".AI7.rCalibration,
            rDiv := "SS1_A2_8RTD_AI_Vars".AI7.rDiv,
            rOutput => "SS1_A2_8RTD_AI_Vars".AI7.rValue);
   "AIvars"(rInput := "SS1_A2_8RTD_AI_Vars".AI7.rValue,
            iFuncSystem := "SS1_A2_8RTD_AI_Vars".AI7.cFuncSystemID,
            iFuncVar := "SS1_A2_8RTD_AI_Vars".AI7.cFuncVar);
END_REGION

REGION Network 8
   RUNG wire#powerrail
      "RTDadv"(iInput := "AI11.02.08", rFilterValue := "SS1_A2_8RTD_AI_Vars".AI8.rFilterSet, rCalibration := "SS1_A2_8RTD_AI_Vars".AI8.rCalibration, rDiv := "SS1_A2_8RTD_AI_Vars".AI8.rDiv, rOutput => "SS1_A2_8RTD_AI_Vars".AI8.rValue)
   END_RUNG
   RUNG wire#powerrail
      "AIvars"(rInput := "SS1_A2_8RTD_AI_Vars".AI8.rValue, iFuncSystem := "SS1_A2_8RTD_AI_Vars".AI8.cFuncSystemID, iFuncVar := "SS1_A2_8RTD_AI_Vars".AI8.cFuncVar)
   END_RUNG
   // the same network as SCL:
   "RTDadv"(iInput := "AI11.02.08",
            rFilterValue := "SS1_A2_8RTD_AI_Vars".AI8.rFilterSet,
            rCalibration := "SS1_A2_8RTD_AI_Vars".AI8.rCalibration,
            rDiv := "SS1_A2_8RTD_AI_Vars".AI8.rDiv,
            rOutput => "SS1_A2_8RTD_AI_Vars".AI8.rValue);
   "AIvars"(rInput := "SS1_A2_8RTD_AI_Vars".AI8.rValue,
            iFuncSystem := "SS1_A2_8RTD_AI_Vars".AI8.cFuncSystemID,
            iFuncVar := "SS1_A2_8RTD_AI_Vars".AI8.cFuncVar);
END_REGION
END_FUNCTION

FUNCTION "SS1_A3_8AI_IO_Update" : Void   // FC11030, LAD
{ S7_Optimized_Access := 'TRUE' }
VERSION : 0.1
// stored: AutoNumber false, IsIECCheckEnabled false, SetENOAutomatically false, UDAEnableTagReadback false
BEGIN

REGION Network 1: AI0
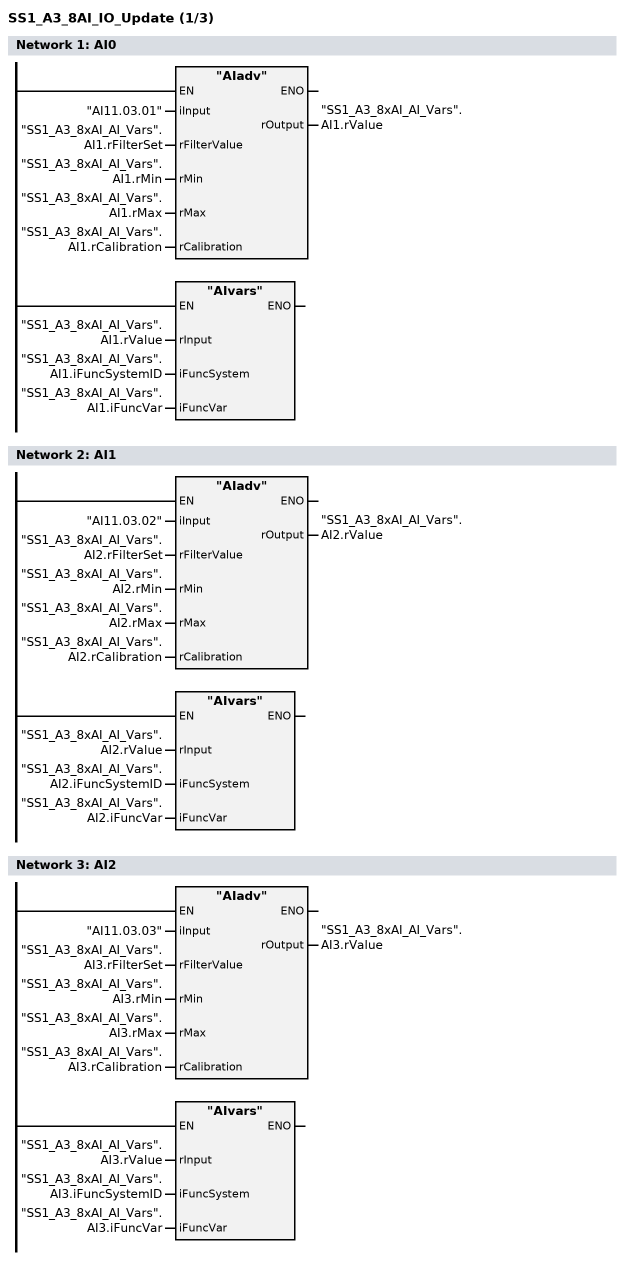
   RUNG wire#powerrail
      "AIadv"(iInput := "AI11.03.01", rFilterValue := "SS1_A3_8xAI_AI_Vars".AI1.rFilterSet, rMin := "SS1_A3_8xAI_AI_Vars".AI1.rMin, rMax := "SS1_A3_8xAI_AI_Vars".AI1.rMax, rCalibration := "SS1_A3_8xAI_AI_Vars".AI1.rCalibration, rOutput => "SS1_A3_8xAI_AI_Vars".AI1.rValue)
   END_RUNG
   RUNG wire#powerrail
      "AIvars"(rInput := "SS1_A3_8xAI_AI_Vars".AI1.rValue, iFuncSystem := "SS1_A3_8xAI_AI_Vars".AI1.iFuncSystemID, iFuncVar := "SS1_A3_8xAI_AI_Vars".AI1.iFuncVar)
   END_RUNG
   // the same network as SCL:
   "AIadv"(iInput := "AI11.03.01",
           rFilterValue := "SS1_A3_8xAI_AI_Vars".AI1.rFilterSet,
           rMin := "SS1_A3_8xAI_AI_Vars".AI1.rMin,
           rMax := "SS1_A3_8xAI_AI_Vars".AI1.rMax,
           rCalibration := "SS1_A3_8xAI_AI_Vars".AI1.rCalibration,
           rOutput => "SS1_A3_8xAI_AI_Vars".AI1.rValue);
   "AIvars"(rInput := "SS1_A3_8xAI_AI_Vars".AI1.rValue,
            iFuncSystem := "SS1_A3_8xAI_AI_Vars".AI1.iFuncSystemID,
            iFuncVar := "SS1_A3_8xAI_AI_Vars".AI1.iFuncVar);
END_REGION

REGION Network 2: AI1
   RUNG wire#powerrail
      "AIadv"(iInput := "AI11.03.02", rFilterValue := "SS1_A3_8xAI_AI_Vars".AI2.rFilterSet, rMin := "SS1_A3_8xAI_AI_Vars".AI2.rMin, rMax := "SS1_A3_8xAI_AI_Vars".AI2.rMax, rCalibration := "SS1_A3_8xAI_AI_Vars".AI2.rCalibration, rOutput => "SS1_A3_8xAI_AI_Vars".AI2.rValue)
   END_RUNG
   RUNG wire#powerrail
      "AIvars"(rInput := "SS1_A3_8xAI_AI_Vars".AI2.rValue, iFuncSystem := "SS1_A3_8xAI_AI_Vars".AI2.iFuncSystemID, iFuncVar := "SS1_A3_8xAI_AI_Vars".AI2.iFuncVar)
   END_RUNG
   // the same network as SCL:
   "AIadv"(iInput := "AI11.03.02",
           rFilterValue := "SS1_A3_8xAI_AI_Vars".AI2.rFilterSet,
           rMin := "SS1_A3_8xAI_AI_Vars".AI2.rMin,
           rMax := "SS1_A3_8xAI_AI_Vars".AI2.rMax,
           rCalibration := "SS1_A3_8xAI_AI_Vars".AI2.rCalibration,
           rOutput => "SS1_A3_8xAI_AI_Vars".AI2.rValue);
   "AIvars"(rInput := "SS1_A3_8xAI_AI_Vars".AI2.rValue,
            iFuncSystem := "SS1_A3_8xAI_AI_Vars".AI2.iFuncSystemID,
            iFuncVar := "SS1_A3_8xAI_AI_Vars".AI2.iFuncVar);
END_REGION

REGION Network 3: AI2
   RUNG wire#powerrail
      "AIadv"(iInput := "AI11.03.03", rFilterValue := "SS1_A3_8xAI_AI_Vars".AI3.rFilterSet, rMin := "SS1_A3_8xAI_AI_Vars".AI3.rMin, rMax := "SS1_A3_8xAI_AI_Vars".AI3.rMax, rCalibration := "SS1_A3_8xAI_AI_Vars".AI3.rCalibration, rOutput => "SS1_A3_8xAI_AI_Vars".AI3.rValue)
   END_RUNG
   RUNG wire#powerrail
      "AIvars"(rInput := "SS1_A3_8xAI_AI_Vars".AI3.rValue, iFuncSystem := "SS1_A3_8xAI_AI_Vars".AI3.iFuncSystemID, iFuncVar := "SS1_A3_8xAI_AI_Vars".AI3.iFuncVar)
   END_RUNG
   // the same network as SCL:
   "AIadv"(iInput := "AI11.03.03",
           rFilterValue := "SS1_A3_8xAI_AI_Vars".AI3.rFilterSet,
           rMin := "SS1_A3_8xAI_AI_Vars".AI3.rMin,
           rMax := "SS1_A3_8xAI_AI_Vars".AI3.rMax,
           rCalibration := "SS1_A3_8xAI_AI_Vars".AI3.rCalibration,
           rOutput => "SS1_A3_8xAI_AI_Vars".AI3.rValue);
   "AIvars"(rInput := "SS1_A3_8xAI_AI_Vars".AI3.rValue,
            iFuncSystem := "SS1_A3_8xAI_AI_Vars".AI3.iFuncSystemID,
            iFuncVar := "SS1_A3_8xAI_AI_Vars".AI3.iFuncVar);
END_REGION

